      movel([0.391008, -1.437717, -2.526713, -0.747959, 1.570796, 1.961804],accel_mss,speed_ms,0,blend_radius_m)
      movel([0.391013, -1.437236, -2.527093, -0.748060, 1.570796, 1.961809],accel_mss,speed_ms,0,blend_radius_m)
      movel([0.391046, -1.436198, -2.527912, -0.748279, 1.570796, 1.961842],accel_mss,speed_ms,0,blend_radius_m)
      movel([0.391091, -1.435157, -2.528733, -0.748500, 1.570796, 1.961887],accel_mss,speed_ms,0,blend_radius_m)
      movel([0.391149, -1.434110, -2.529556, -0.748724, 1.570796, 1.961945],accel_mss,speed_ms,0,blend_radius_m)
      movel([0.391230, -1.432906, -2.530500, -0.748983, 1.570796, 1.962026],accel_mss,speed_ms,0,blend_radius_m)
      movel([0.391323, -1.431698, -2.531445, -0.749246, 1.570796, 1.962119],accel_mss,speed_ms,0,blend_radius_m)
      movel([0.391429, -1.430482, -2.532395, -0.749512, 1.570796, 1.962226],accel_mss,speed_ms,0,blend_radius_m)
      movel([0.391551, -1.429259, -2.533347, -0.749782, 1.570796, 1.962348],accel_mss,speed_ms,0,blend_radius_m)
      movel([0.391688, -1.428032, -2.534301, -0.750056, 1.570796, 1.962484],accel_mss,speed_ms,0,blend_radius_m)
      movel([0.391837, -1.426799, -2.535257, -0.750333, 1.570796, 1.962634],accel_mss,speed_ms,0,blend_radius_m)
      movel([0.392000, -1.425405, -2.536335, -0.750649, 1.570796, 1.962797],accel_mss,speed_ms,0,blend_radius_m)
      movel([0.392135, -1.424015, -2.537407, -0.750967, 1.570796, 1.962931],accel_mss,speed_ms,0,blend_radius_m)
      movel([0.392245, -1.422628, -2.538474, -0.751287, 1.570796, 1.963042],accel_mss,speed_ms,0,blend_radius_m)
      movel([0.392325, -1.421249, -2.539532, -0.751608, 1.570796, 1.963121],accel_mss,speed_ms,0,blend_radius_m)
      movel([0.392346, -1.420560, -2.540059, -0.751770, 1.570796, 1.963143],accel_mss,speed_ms,0,blend_radius_m)
      movel([0.392346, -1.419880, -2.540579, -0.751930, 1.570796, 1.963143],accel_mss,speed_ms,0,blend_radius_m)
      movel([0.392325, -1.419207, -2.541092, -0.752089, 1.570796, 1.963121],accel_mss,speed_ms,0,blend_radius_m)
      movel([0.392281, -1.418541, -2.541601, -0.752247, 1.570796, 1.963077],accel_mss,speed_ms,0,blend_radius_m)
      movel([0.392215, -1.417882, -2.542102, -0.752405, 1.570796, 1.963012],accel_mss,speed_ms,0,blend_radius_m)
      movel([0.392127, -1.417234, -2.542595, -0.752560, 1.570796, 1.962924],accel_mss,speed_ms,0,blend_radius_m)
      movel([0.392031, -1.416697, -2.543003, -0.752689, 1.570796, 1.962828],accel_mss,speed_ms,0,blend_radius_m)
      movel([0.391914, -1.416172, -2.543402, -0.752815, 1.570796, 1.962711],accel_mss,speed_ms,0,blend_radius_m)
      movel([0.391773, -1.415658, -2.543791, -0.752940, 1.570796, 1.962569],accel_mss,speed_ms,0,blend_radius_m)
      movel([0.391607, -1.415156, -2.544171, -0.753062, 1.570796, 1.962404],accel_mss,speed_ms,0,blend_radius_m)
      movel([0.391419, -1.414665, -2.544543, -0.753181, 1.570796, 1.962216],accel_mss,speed_ms,0,blend_radius_m)
      movel([0.391209, -1.414190, -2.544902, -0.753297, 1.570796, 1.962005],accel_mss,speed_ms,0,blend_radius_m)
      movel([0.390979, -1.413733, -2.545247, -0.753409, 1.570796, 1.961776],accel_mss,speed_ms,0,blend_radius_m)
      movel([0.390725, -1.413291, -2.545580, -0.753517, 1.570796, 1.961521],accel_mss,speed_ms,0,blend_radius_m)
      movel([0.390449, -1.412863, -2.545903, -0.753623, 1.570796, 1.961245],accel_mss,speed_ms,0,blend_radius_m)
      movel([0.390149, -1.412454, -2.546211, -0.753724, 1.570796, 1.960945],accel_mss,speed_ms,0,blend_radius_m)
      movel([0.389829, -1.412060, -2.546508, -0.753821, 1.570796, 1.960625],accel_mss,speed_ms,0,blend_radius_m)
      movel([0.389486, -1.411681, -2.546793, -0.753915, 1.570796, 1.960283],accel_mss,speed_ms,0,blend_radius_m)
      movel([0.389035, -1.411243, -2.547122, -0.754024, 1.570796, 1.959831],accel_mss,speed_ms,0,blend_radius_m)
      movel([0.388548, -1.410836, -2.547428, -0.754125, 1.570796, 1.959344],accel_mss,speed_ms,0,blend_radius_m)
      movel([0.388004, -1.410440, -2.547725, -0.754224, 1.570796, 1.958800],accel_mss,speed_ms,0,blend_radius_m)
      movel([0.387428, -1.410075, -2.547998, -0.754316, 1.570796, 1.958225],accel_mss,speed_ms,0,blend_radius_m)
      movel([0.386840, -1.409745, -2.548245, -0.754398, 1.570796, 1.957636],accel_mss,speed_ms,0,blend_radius_m)
      movel([0.386219, -1.409448, -2.548468, -0.754473, 1.570796, 1.957016],accel_mss,speed_ms,0,blend_radius_m)
      movel([0.385828, -1.409285, -2.548590, -0.754514, 1.570796, 1.956624],accel_mss,speed_ms,0,blend_radius_m)
      movel([0.385423, -1.409139, -2.548699, -0.754551, 1.570796, 1.956219],accel_mss,speed_ms,0,blend_radius_m)
      movel([0.385006, -1.409009, -2.548796, -0.754584, 1.570796, 1.955802],accel_mss,speed_ms,0,blend_radius_m)
      movel([0.383851, -1.408685, -2.549039, -0.754665, 1.570796, 1.954647],accel_mss,speed_ms,0,blend_radius_m)
      movel([0.383532, -1.409238, -2.548625, -0.754526, 1.570796, 1.954329],accel_mss,speed_ms,0,blend_radius_m)
      movel([0.383126, -1.409975, -2.548073, -0.754341, 1.570796, 1.953923],accel_mss,speed_ms,0,blend_radius_m)
      movel([0.381046, -1.414103, -2.544967, -0.753318, 1.570796, 1.951842],accel_mss,speed_ms,0,blend_radius_m)
      movel([0.381019, -1.414157, -2.544927, -0.753305, 1.570796, 1.951816],accel_mss,speed_ms,0,blend_radius_m)
      movel([0.380984, -1.414209, -2.544887, -0.753292, 1.570796, 1.951781],accel_mss,speed_ms,0,blend_radius_m)
      movel([0.380941, -1.414259, -2.544850, -0.753280, 1.570796, 1.951738],accel_mss,speed_ms,0,blend_radius_m)
      movel([0.380899, -1.414296, -2.544822, -0.753271, 1.570796, 1.951696],accel_mss,speed_ms,0,blend_radius_m)
      movel([0.380850, -1.414325, -2.544800, -0.753264, 1.570796, 1.951646],accel_mss,speed_ms,0,blend_radius_m)
      movel([0.380798, -1.414343, -2.544787, -0.753260, 1.570796, 1.951594],accel_mss,speed_ms,0,blend_radius_m)
      movel([0.380720, -1.414359, -2.544774, -0.753256, 1.570796, 1.951516],accel_mss,speed_ms,0,blend_radius_m)
      movel([0.380641, -1.414367, -2.544768, -0.753254, 1.570796, 1.951438],accel_mss,speed_ms,0,blend_radius_m)
      movel([0.380568, -1.414366, -2.544769, -0.753254, 1.570796, 1.951365],accel_mss,speed_ms,0,blend_radius_m)
      movel([0.380337, -1.414350, -2.544781, -0.753258, 1.570796, 1.951133],accel_mss,speed_ms,0,blend_radius_m)
      movel([0.380108, -1.414330, -2.544796, -0.753263, 1.570796, 1.950904],accel_mss,speed_ms,0,blend_radius_m)
      movel([0.377696, -1.414133, -2.544945, -0.753311, 1.570796, 1.948493],accel_mss,speed_ms,0,blend_radius_m)
      movel([0.377544, -1.414147, -2.544935, -0.753308, 1.570796, 1.948341],accel_mss,speed_ms,0,blend_radius_m)
      movel([0.377385, -1.414188, -2.544903, -0.753297, 1.570796, 1.948181],accel_mss,speed_ms,0,blend_radius_m)
      movel([0.377316, -1.414222, -2.544878, -0.753289, 1.570796, 1.948112],accel_mss,speed_ms,0,blend_radius_m)
      movel([0.377256, -1.414274, -2.544838, -0.753277, 1.570796, 1.948053],accel_mss,speed_ms,0,blend_radius_m)
      movel([0.377217, -1.414337, -2.544791, -0.753261, 1.570796, 1.948013],accel_mss,speed_ms,0,blend_radius_m)
      movel([0.377159, -1.414466, -2.544693, -0.753230, 1.570796, 1.947956],accel_mss,speed_ms,0,blend_radius_m)
      movel([0.377090, -1.414598, -2.544594, -0.753197, 1.570796, 1.947886],accel_mss,speed_ms,0,blend_radius_m)
      movel([0.377010, -1.414725, -2.544497, -0.753166, 1.570796, 1.947807],accel_mss,speed_ms,0,blend_radius_m)
      movel([0.376921, -1.414851, -2.544402, -0.753136, 1.570796, 1.947717],accel_mss,speed_ms,0,blend_radius_m)
      movel([0.376332, -1.415635, -2.543809, -0.752945, 1.570796, 1.947129],accel_mss,speed_ms,0,blend_radius_m)
      movel([0.375736, -1.416416, -2.543217, -0.752757, 1.570796, 1.946533],accel_mss,speed_ms,0,blend_radius_m)
      movel([0.375083, -1.417257, -2.542578, -0.752554, 1.570796, 1.945880],accel_mss,speed_ms,0,blend_radius_m)
      movel([0.374421, -1.418095, -2.541941, -0.752354, 1.570796, 1.945218],accel_mss,speed_ms,0,blend_radius_m)
      movel([0.373801, -1.418859, -2.541359, -0.752172, 1.570796, 1.944597],accel_mss,speed_ms,0,blend_radius_m)
      movel([0.373169, -1.419616, -2.540781, -0.751993, 1.570796, 1.943965],accel_mss,speed_ms,0,blend_radius_m)
      movel([0.372591, -1.420290, -2.540265, -0.751833, 1.570796, 1.943387],accel_mss,speed_ms,0,blend_radius_m)
      movel([0.372002, -1.420960, -2.539753, -0.751676, 1.570796, 1.942799],accel_mss,speed_ms,0,blend_radius_m)
      movel([0.371402, -1.421622, -2.539246, -0.751521, 1.570796, 1.942199],accel_mss,speed_ms,0,blend_radius_m)
      movel([0.370791, -1.422279, -2.538742, -0.751368, 1.570796, 1.941588],accel_mss,speed_ms,0,blend_radius_m)
      movel([0.370171, -1.422927, -2.538244, -0.751218, 1.570796, 1.940968],accel_mss,speed_ms,0,blend_radius_m)
      movel([0.369539, -1.423568, -2.537751, -0.751070, 1.570796, 1.940336],accel_mss,speed_ms,0,blend_radius_m)
      movel([0.368900, -1.424201, -2.537264, -0.750924, 1.570796, 1.939697],accel_mss,speed_ms,0,blend_radius_m)
      movel([0.368252, -1.424827, -2.536781, -0.750781, 1.570796, 1.939048],accel_mss,speed_ms,0,blend_radius_m)
      movel([0.367591, -1.425445, -2.536304, -0.750640, 1.570796, 1.938388],accel_mss,speed_ms,0,blend_radius_m)
      movel([0.366924, -1.426056, -2.535832, -0.750501, 1.570796, 1.937720],accel_mss,speed_ms,0,blend_radius_m)
      movel([0.366244, -1.426659, -2.535366, -0.750365, 1.570796, 1.937041],accel_mss,speed_ms,0,blend_radius_m)
      movel([0.365557, -1.427255, -2.534904, -0.750230, 1.570796, 1.936354],accel_mss,speed_ms,0,blend_radius_m)
      movel([0.364862, -1.427840, -2.534450, -0.750099, 1.570796, 1.935659],accel_mss,speed_ms,0,blend_radius_m)
      movel([0.364160, -1.428418, -2.534002, -0.749970, 1.570796, 1.934957],accel_mss,speed_ms,0,blend_radius_m)
      movel([0.363449, -1.428986, -2.533560, -0.749843, 1.570796, 1.934245],accel_mss,speed_ms,0,blend_radius_m)
      movel([0.362732, -1.429545, -2.533125, -0.749719, 1.570796, 1.933528],accel_mss,speed_ms,0,blend_radius_m)
      movel([0.362008, -1.430092, -2.532699, -0.749598, 1.570796, 1.932805],accel_mss,speed_ms,0,blend_radius_m)
      movel([0.361278, -1.430632, -2.532278, -0.749479, 1.570796, 1.932074],accel_mss,speed_ms,0,blend_radius_m)
      movel([0.360551, -1.431154, -2.531870, -0.749364, 1.570796, 1.931347],accel_mss,speed_ms,0,blend_radius_m)
      movel([0.359817, -1.431667, -2.531470, -0.749252, 1.570796, 1.930614],accel_mss,speed_ms,0,blend_radius_m)
      movel([0.359077, -1.432169, -2.531077, -0.749143, 1.570796, 1.929874],accel_mss,speed_ms,0,blend_radius_m)
      movel([0.358332, -1.432660, -2.530693, -0.749036, 1.570796, 1.929128],accel_mss,speed_ms,0,blend_radius_m)
      movel([0.357582, -1.433140, -2.530317, -0.748932, 1.570796, 1.928379],accel_mss,speed_ms,0,blend_radius_m)
      movel([0.356828, -1.433611, -2.529947, -0.748831, 1.570796, 1.927625],accel_mss,speed_ms,0,blend_radius_m)
      movel([0.356069, -1.434070, -2.529587, -0.748732, 1.570796, 1.926865],accel_mss,speed_ms,0,blend_radius_m)
      movel([0.355306, -1.434516, -2.529236, -0.748636, 1.570796, 1.926102],accel_mss,speed_ms,0,blend_radius_m)
      movel([0.354537, -1.434953, -2.528893, -0.748543, 1.570796, 1.925333],accel_mss,speed_ms,0,blend_radius_m)
      movel([0.353788, -1.435366, -2.528568, -0.748455, 1.570796, 1.924585],accel_mss,speed_ms,0,blend_radius_m)
      movel([0.353034, -1.435767, -2.528252, -0.748370, 1.570796, 1.923830],accel_mss,speed_ms,0,blend_radius_m)
      movel([0.352277, -1.436154, -2.527947, -0.748288, 1.570796, 1.923073],accel_mss,speed_ms,0,blend_radius_m)
      movel([0.351516, -1.436531, -2.527649, -0.748208, 1.570796, 1.922312],accel_mss,speed_ms,0,blend_radius_m)
      movel([0.350754, -1.436894, -2.527363, -0.748132, 1.570796, 1.921551],accel_mss,speed_ms,0,blend_radius_m)
      movel([0.349988, -1.437243, -2.527088, -0.748058, 1.570796, 1.920784],accel_mss,speed_ms,0,blend_radius_m)
      movel([0.349222, -1.437580, -2.526821, -0.747988, 1.570796, 1.920018],accel_mss,speed_ms,0,blend_radius_m)
      movel([0.348452, -1.437905, -2.526565, -0.747920, 1.570796, 1.919249],accel_mss,speed_ms,0,blend_radius_m)
      movel([0.347682, -1.438215, -2.526319, -0.747855, 1.570796, 1.918479],accel_mss,speed_ms,0,blend_radius_m)
      movel([0.346942, -1.438501, -2.526093, -0.747796, 1.570796, 1.917738],accel_mss,speed_ms,0,blend_radius_m)
      movel([0.346197, -1.438776, -2.525874, -0.747738, 1.570796, 1.916993],accel_mss,speed_ms,0,blend_radius_m)
      movel([0.345456, -1.439037, -2.525667, -0.747684, 1.570796, 1.916252],accel_mss,speed_ms,0,blend_radius_m)
      movel([0.344712, -1.439289, -2.525468, -0.747632, 1.570796, 1.915508],accel_mss,speed_ms,0,blend_radius_m)
      movel([0.343967, -1.439527, -2.525279, -0.747583, 1.570796, 1.914764],accel_mss,speed_ms,0,blend_radius_m)
      movel([0.343243, -1.439745, -2.525106, -0.747538, 1.570796, 1.914040],accel_mss,speed_ms,0,blend_radius_m)
      movel([0.342517, -1.439952, -2.524941, -0.747495, 1.570796, 1.913314],accel_mss,speed_ms,0,blend_radius_m)
      movel([0.341795, -1.440145, -2.524788, -0.747456, 1.570796, 1.912591],accel_mss,speed_ms,0,blend_radius_m)
      movel([0.341071, -1.440326, -2.524644, -0.747419, 1.570796, 1.911867],accel_mss,speed_ms,0,blend_radius_m)
      movel([0.340352, -1.440493, -2.524512, -0.747384, 1.570796, 1.911149],accel_mss,speed_ms,0,blend_radius_m)
      movel([0.339621, -1.440649, -2.524388, -0.747352, 1.570796, 1.910417],accel_mss,speed_ms,0,blend_radius_m)
      movel([0.338890, -1.440790, -2.524275, -0.747323, 1.570796, 1.909687],accel_mss,speed_ms,0,blend_radius_m)
      movel([0.338165, -1.440920, -2.524172, -0.747297, 1.570796, 1.908961],accel_mss,speed_ms,0,blend_radius_m)
      movel([0.337442, -1.441036, -2.524080, -0.747273, 1.570796, 1.908238],accel_mss,speed_ms,0,blend_radius_m)
      movel([0.336723, -1.441138, -2.523999, -0.747252, 1.570796, 1.907519],accel_mss,speed_ms,0,blend_radius_m)
      movel([0.335963, -1.441234, -2.523922, -0.747233, 1.570796, 1.906759],accel_mss,speed_ms,0,blend_radius_m)
      movel([0.335208, -1.441316, -2.523857, -0.747216, 1.570796, 1.906004],accel_mss,speed_ms,0,blend_radius_m)
      movel([0.334457, -1.441386, -2.523801, -0.747202, 1.570796, 1.905253],accel_mss,speed_ms,0,blend_radius_m)
      movel([0.333710, -1.441447, -2.523753, -0.747189, 1.570796, 1.904507],accel_mss,speed_ms,0,blend_radius_m)
      movel([0.332967, -1.441493, -2.523716, -0.747180, 1.570796, 1.903763],accel_mss,speed_ms,0,blend_radius_m)
      movel([0.329715, -1.441675, -2.523571, -0.747143, 1.570796, 1.900511],accel_mss,speed_ms,0,blend_radius_m)
      movel([0.329386, -1.442137, -2.523203, -0.747049, 1.570796, 1.900182],accel_mss,speed_ms,0,blend_radius_m)
      movel([0.329307, -1.442240, -2.523121, -0.747029, 1.570796, 1.900104],accel_mss,speed_ms,0,blend_radius_m)
      movel([0.329218, -1.442336, -2.523044, -0.747009, 1.570796, 1.900015],accel_mss,speed_ms,0,blend_radius_m)
      movel([0.329123, -1.442425, -2.522973, -0.746991, 1.570796, 1.899919],accel_mss,speed_ms,0,blend_radius_m)
      movel([0.329019, -1.442510, -2.522905, -0.746974, 1.570796, 1.899815],accel_mss,speed_ms,0,blend_radius_m)
      movel([0.328913, -1.442580, -2.522849, -0.746960, 1.570796, 1.899710],accel_mss,speed_ms,0,blend_radius_m)
      movel([0.328802, -1.442642, -2.522799, -0.746947, 1.570796, 1.899598],accel_mss,speed_ms,0,blend_radius_m)
      movel([0.328694, -1.442690, -2.522761, -0.746938, 1.570796, 1.899490],accel_mss,speed_ms,0,blend_radius_m)
      movel([0.328584, -1.442725, -2.522734, -0.746931, 1.570796, 1.899380],accel_mss,speed_ms,0,blend_radius_m)
      movel([0.328442, -1.442758, -2.522707, -0.746924, 1.570796, 1.899238],accel_mss,speed_ms,0,blend_radius_m)
      movel([0.328305, -1.442780, -2.522690, -0.746920, 1.570796, 1.899101],accel_mss,speed_ms,0,blend_radius_m)
      movel([0.328168, -1.442793, -2.522679, -0.746917, 1.570796, 1.898964],accel_mss,speed_ms,0,blend_radius_m)
      movel([0.328036, -1.442794, -2.522678, -0.746917, 1.570796, 1.898832],accel_mss,speed_ms,0,blend_radius_m)
      movel([0.323844, -1.442695, -2.522758, -0.746937, 1.570796, 1.894641],accel_mss,speed_ms,0,blend_radius_m)
      movel([0.321918, -1.442649, -2.522794, -0.746946, 1.570796, 1.892714],accel_mss,speed_ms,0,blend_radius_m)
      movel([0.319994, -1.442597, -2.522836, -0.746956, 1.570796, 1.890790],accel_mss,speed_ms,0,blend_radius_m)
      movel([0.319329, -1.442571, -2.522856, -0.746962, 1.570796, 1.890125],accel_mss,speed_ms,0,blend_radius_m)
      movel([0.318669, -1.442535, -2.522885, -0.746969, 1.570796, 1.889465],accel_mss,speed_ms,0,blend_radius_m)
      movel([0.318013, -1.442490, -2.522921, -0.746978, 1.570796, 1.888809],accel_mss,speed_ms,0,blend_radius_m)
      movel([0.317850, -1.442468, -2.522939, -0.746983, 1.570796, 1.888646],accel_mss,speed_ms,0,blend_radius_m)
      movel([0.317697, -1.442429, -2.522970, -0.746990, 1.570796, 1.888493],accel_mss,speed_ms,0,blend_radius_m)
      movel([0.317553, -1.442377, -2.523011, -0.747001, 1.570796, 1.888349],accel_mss,speed_ms,0,blend_radius_m)
      movel([0.317424, -1.442309, -2.523065, -0.747015, 1.570796, 1.888220],accel_mss,speed_ms,0,blend_radius_m)
      movel([0.317355, -1.442253, -2.523110, -0.747026, 1.570796, 1.888151],accel_mss,speed_ms,0,blend_radius_m)
      movel([0.317298, -1.442186, -2.523163, -0.747039, 1.570796, 1.888095],accel_mss,speed_ms,0,blend_radius_m)
      movel([0.317262, -1.442106, -2.523227, -0.747056, 1.570796, 1.888058],accel_mss,speed_ms,0,blend_radius_m)
      movel([0.317241, -1.442017, -2.523299, -0.747074, 1.570796, 1.888038],accel_mss,speed_ms,0,blend_radius_m)
      movel([0.317241, -1.441920, -2.523376, -0.747093, 1.570796, 1.888037],accel_mss,speed_ms,0,blend_radius_m)
      movel([0.317266, -1.441727, -2.523529, -0.747133, 1.570796, 1.888062],accel_mss,speed_ms,0,blend_radius_m)
      movel([0.317307, -1.441531, -2.523686, -0.747172, 1.570796, 1.888103],accel_mss,speed_ms,0,blend_radius_m)
      movel([0.317366, -1.441332, -2.523844, -0.747213, 1.570796, 1.888162],accel_mss,speed_ms,0,blend_radius_m)
      movel([0.317441, -1.441131, -2.524004, -0.747254, 1.570796, 1.888237],accel_mss,speed_ms,0,blend_radius_m)
      movel([0.317857, -1.440156, -2.524779, -0.747453, 1.570796, 1.888653],accel_mss,speed_ms,0,blend_radius_m)
      movel([0.318288, -1.439181, -2.525553, -0.747655, 1.570796, 1.889084],accel_mss,speed_ms,0,blend_radius_m)
      movel([0.319674, -1.435971, -2.528092, -0.748327, 1.570796, 1.890471],accel_mss,speed_ms,0,blend_radius_m)
      movel([0.319898, -1.435346, -2.528583, -0.748459, 1.570796, 1.890694],accel_mss,speed_ms,0,blend_radius_m)
      movel([0.318917, -1.435409, -2.528534, -0.748446, 1.570796, 1.889714],accel_mss,speed_ms,0,blend_radius_m)
      movel([0.317936, -1.435473, -2.528483, -0.748432, 1.570796, 1.888733],accel_mss,speed_ms,0,blend_radius_m)
      movel([0.315692, -1.441850, -2.523431, -0.747108, 1.570796, 1.886489],accel_mss,speed_ms,0,blend_radius_m)
      movel([0.314773, -1.444460, -2.521346, -0.746583, 1.570796, 1.885569],accel_mss,speed_ms,0,blend_radius_m)
      movel([0.313846, -1.447061, -2.519257, -0.746071, 1.570796, 1.884642],accel_mss,speed_ms,0,blend_radius_m)
      movel([0.313754, -1.447292, -2.519071, -0.746026, 1.570796, 1.884550],accel_mss,speed_ms,0,blend_radius_m)
      movel([0.313650, -1.447523, -2.518885, -0.745981, 1.570796, 1.884446],accel_mss,speed_ms,0,blend_radius_m)
      movel([0.313528, -1.447754, -2.518699, -0.745936, 1.570796, 1.884325],accel_mss,speed_ms,0,blend_radius_m)
      movel([0.313393, -1.447983, -2.518515, -0.745892, 1.570796, 1.884189],accel_mss,speed_ms,0,blend_radius_m)
      movel([0.313241, -1.448208, -2.518333, -0.745848, 1.570796, 1.884037],accel_mss,speed_ms,0,blend_radius_m)
      movel([0.313169, -1.448302, -2.518257, -0.745830, 1.570796, 1.883966],accel_mss,speed_ms,0,blend_radius_m)
      movel([0.313084, -1.448391, -2.518185, -0.745813, 1.570796, 1.883881],accel_mss,speed_ms,0,blend_radius_m)
      movel([0.312991, -1.448475, -2.518117, -0.745797, 1.570796, 1.883787],accel_mss,speed_ms,0,blend_radius_m)
      movel([0.312890, -1.448550, -2.518057, -0.745782, 1.570796, 1.883686],accel_mss,speed_ms,0,blend_radius_m)
      movel([0.312781, -1.448614, -2.518005, -0.745770, 1.570796, 1.883577],accel_mss,speed_ms,0,blend_radius_m)
      movel([0.312669, -1.448670, -2.517960, -0.745759, 1.570796, 1.883466],accel_mss,speed_ms,0,blend_radius_m)
      movel([0.312558, -1.448711, -2.517927, -0.745751, 1.570796, 1.883355],accel_mss,speed_ms,0,blend_radius_m)
      movel([0.312444, -1.448742, -2.517902, -0.745745, 1.570796, 1.883241],accel_mss,speed_ms,0,blend_radius_m)
      movel([0.312092, -1.448811, -2.517846, -0.745732, 1.570796, 1.882888],accel_mss,speed_ms,0,blend_radius_m)
      movel([0.311740, -1.448872, -2.517797, -0.745720, 1.570796, 1.882536],accel_mss,speed_ms,0,blend_radius_m)
      movel([0.311392, -1.448920, -2.517758, -0.745711, 1.570796, 1.882188],accel_mss,speed_ms,0,blend_radius_m)
      movel([0.311046, -1.448959, -2.517726, -0.745704, 1.570796, 1.881842],accel_mss,speed_ms,0,blend_radius_m)
      movel([0.310704, -1.448986, -2.517705, -0.745698, 1.570796, 1.881500],accel_mss,speed_ms,0,blend_radius_m)
      movel([0.308856, -1.449110, -2.517604, -0.745675, 1.570796, 1.879653],accel_mss,speed_ms,0,blend_radius_m)
      movel([0.307890, -1.451920, -2.515327, -0.745142, 1.570796, 1.878686],accel_mss,speed_ms,0,blend_radius_m)
      movel([0.306930, -1.454717, -2.513049, -0.744623, 1.570796, 1.877726],accel_mss,speed_ms,0,blend_radius_m)
      movel([0.321643, -1.458076, -2.510297, -0.744016, 1.570796, 1.892440],accel_mss,speed_ms,0,blend_radius_m)
      movel([0.327249, -1.459428, -2.509184, -0.743777, 1.570796, 1.898045],accel_mss,speed_ms,0,blend_radius_m)
      movel([0.331985, -1.460602, -2.508216, -0.743571, 1.570796, 1.902781],accel_mss,speed_ms,0,blend_radius_m)
      movel([0.336201, -1.461671, -2.507332, -0.743386, 1.570796, 1.906997],accel_mss,speed_ms,0,blend_radius_m)
      movel([0.336481, -1.461719, -2.507292, -0.743378, 1.570796, 1.907277],accel_mss,speed_ms,0,blend_radius_m)
      movel([0.336565, -1.461686, -2.507319, -0.743383, 1.570796, 1.907361],accel_mss,speed_ms,0,blend_radius_m)
      movel([0.336663, -1.461615, -2.507378, -0.743396, 1.570796, 1.907460],accel_mss,speed_ms,0,blend_radius_m)
      movel([0.336752, -1.461531, -2.507448, -0.743410, 1.570796, 1.907549],accel_mss,speed_ms,0,blend_radius_m)
      movel([0.336997, -1.461218, -2.507707, -0.743464, 1.570796, 1.907793],accel_mss,speed_ms,0,blend_radius_m)
      movel([0.337381, -1.460630, -2.508193, -0.743566, 1.570796, 1.908177],accel_mss,speed_ms,0,blend_radius_m)
      movel([0.337671, -1.460183, -2.508561, -0.743644, 1.570796, 1.908467],accel_mss,speed_ms,0,blend_radius_m)
      movel([0.337804, -1.459986, -2.508724, -0.743679, 1.570796, 1.908601],accel_mss,speed_ms,0,blend_radius_m)
      movel([0.337943, -1.459793, -2.508883, -0.743713, 1.570796, 1.908739],accel_mss,speed_ms,0,blend_radius_m)
      movel([0.338182, -1.459473, -2.509147, -0.743769, 1.570796, 1.908978],accel_mss,speed_ms,0,blend_radius_m)
      movel([0.338208, -1.459442, -2.509172, -0.743774, 1.570796, 1.909005],accel_mss,speed_ms,0,blend_radius_m)
      movel([0.338242, -1.459415, -2.509195, -0.743779, 1.570796, 1.909038],accel_mss,speed_ms,0,blend_radius_m)
      movel([0.338277, -1.459394, -2.509212, -0.743783, 1.570796, 1.909074],accel_mss,speed_ms,0,blend_radius_m)
      movel([0.338400, -1.459338, -2.509258, -0.743793, 1.570796, 1.909197],accel_mss,speed_ms,0,blend_radius_m)
      movel([0.338523, -1.459294, -2.509295, -0.743800, 1.570796, 1.909319],accel_mss,speed_ms,0,blend_radius_m)
      movel([0.338648, -1.459260, -2.509323, -0.743807, 1.570796, 1.909445],accel_mss,speed_ms,0,blend_radius_m)
      movel([0.343772, -1.458166, -2.510223, -0.744000, 1.570796, 1.914568],accel_mss,speed_ms,0,blend_radius_m)
      movel([0.348794, -1.457117, -2.511085, -0.744188, 1.570796, 1.919590],accel_mss,speed_ms,0,blend_radius_m)
      movel([0.348995, -1.457081, -2.511114, -0.744194, 1.570796, 1.919791],accel_mss,speed_ms,0,blend_radius_m)
      movel([0.349193, -1.457058, -2.511133, -0.744198, 1.570796, 1.919989],accel_mss,speed_ms,0,blend_radius_m)
      movel([0.349389, -1.457046, -2.511142, -0.744200, 1.570796, 1.920185],accel_mss,speed_ms,0,blend_radius_m)
      movel([0.349479, -1.457050, -2.511140, -0.744200, 1.570796, 1.920275],accel_mss,speed_ms,0,blend_radius_m)
      movel([0.349560, -1.457063, -2.511128, -0.744197, 1.570796, 1.920357],accel_mss,speed_ms,0,blend_radius_m)
      movel([0.349638, -1.457089, -2.511107, -0.744193, 1.570796, 1.920434],accel_mss,speed_ms,0,blend_radius_m)
      movel([0.351833, -1.458041, -2.510325, -0.744022, 1.570796, 1.922629],accel_mss,speed_ms,0,blend_radius_m)
      movel([0.353078, -1.458589, -2.509875, -0.743925, 1.570796, 1.923875],accel_mss,speed_ms,0,blend_radius_m)
      movel([0.354315, -1.459145, -2.509417, -0.743827, 1.570796, 1.925111],accel_mss,speed_ms,0,blend_radius_m)
      movel([0.355751, -1.459804, -2.508874, -0.743711, 1.570796, 1.926547],accel_mss,speed_ms,0,blend_radius_m)
      movel([0.357181, -1.460468, -2.508327, -0.743595, 1.570796, 1.927977],accel_mss,speed_ms,0,blend_radius_m)
      movel([0.364532, -1.463955, -2.505438, -0.742996, 1.570796, 1.935329],accel_mss,speed_ms,0,blend_radius_m)
      movel([0.364147, -1.464542, -2.504950, -0.742897, 1.570796, 1.934944],accel_mss,speed_ms,0,blend_radius_m)
      movel([0.360132, -1.470721, -2.499780, -0.741888, 1.570796, 1.930928],accel_mss,speed_ms,0,blend_radius_m)
      movel([0.359272, -1.472034, -2.498674, -0.741681, 1.570796, 1.930068],accel_mss,speed_ms,0,blend_radius_m)
      movel([0.358506, -1.473198, -2.497691, -0.741500, 1.570796, 1.929302],accel_mss,speed_ms,0,blend_radius_m)
      movel([0.358478, -1.473230, -2.497664, -0.741495, 1.570796, 1.929275],accel_mss,speed_ms,0,blend_radius_m)
      movel([0.358446, -1.473258, -2.497641, -0.741491, 1.570796, 1.929243],accel_mss,speed_ms,0,blend_radius_m)
      movel([0.358424, -1.473268, -2.497632, -0.741489, 1.570796, 1.929220],accel_mss,speed_ms,0,blend_radius_m)
      movel([0.358402, -1.473270, -2.497630, -0.741489, 1.570796, 1.929198],accel_mss,speed_ms,0,blend_radius_m)
      movel([0.358383, -1.473264, -2.497635, -0.741490, 1.570796, 1.929179],accel_mss,speed_ms,0,blend_radius_m)
      movel([0.357147, -1.472418, -2.498350, -0.741621, 1.570796, 1.927943],accel_mss,speed_ms,0,blend_radius_m)
      movel([0.356454, -1.471942, -2.498752, -0.741695, 1.570796, 1.927250],accel_mss,speed_ms,0,blend_radius_m)
      movel([0.355765, -1.471462, -2.499156, -0.741771, 1.570796, 1.926561],accel_mss,speed_ms,0,blend_radius_m)
      movel([0.354136, -1.470317, -2.500120, -0.741952, 1.570796, 1.924932],accel_mss,speed_ms,0,blend_radius_m)
      movel([0.352498, -1.469178, -2.501076, -0.742134, 1.570796, 1.923294],accel_mss,speed_ms,0,blend_radius_m)
      movel([0.351087, -1.468242, -2.501862, -0.742286, 1.570796, 1.921883],accel_mss,speed_ms,0,blend_radius_m)
      movel([0.349797, -1.467428, -2.502543, -0.742418, 1.570796, 1.920593],accel_mss,speed_ms,0,blend_radius_m)
      movel([0.349754, -1.467437, -2.502535, -0.742417, 1.570796, 1.920550],accel_mss,speed_ms,0,blend_radius_m)
      movel([0.349713, -1.467460, -2.502516, -0.742413, 1.570796, 1.920510],accel_mss,speed_ms,0,blend_radius_m)
      movel([0.349617, -1.467544, -2.502445, -0.742399, 1.570796, 1.920413],accel_mss,speed_ms,0,blend_radius_m)
      movel([0.349532, -1.467639, -2.502366, -0.742384, 1.570796, 1.920328],accel_mss,speed_ms,0,blend_radius_m)
      movel([0.349462, -1.467739, -2.502282, -0.742367, 1.570796, 1.920258],accel_mss,speed_ms,0,blend_radius_m)
      movel([0.344256, -1.476421, -2.494959, -0.741009, 1.570796, 1.915053],accel_mss,speed_ms,0,blend_radius_m)
      movel([0.344252, -1.476475, -2.494912, -0.741001, 1.570796, 1.915048],accel_mss,speed_ms,0,blend_radius_m)
      movel([0.344270, -1.476520, -2.494875, -0.740995, 1.570796, 1.915067],accel_mss,speed_ms,0,blend_radius_m)
      movel([0.344294, -1.476539, -2.494859, -0.740992, 1.570796, 1.915091],accel_mss,speed_ms,0,blend_radius_m)
      movel([0.344333, -1.476539, -2.494858, -0.740992, 1.570796, 1.915130],accel_mss,speed_ms,0,blend_radius_m)
      movel([0.348677, -1.475673, -2.495594, -0.741122, 1.570796, 1.919474],accel_mss,speed_ms,0,blend_radius_m)
      movel([0.353320, -1.474728, -2.496396, -0.741265, 1.570796, 1.924117],accel_mss,speed_ms,0,blend_radius_m)
      movel([0.355242, -1.474345, -2.496720, -0.741323, 1.570796, 1.926039],accel_mss,speed_ms,0,blend_radius_m)
      movel([0.356189, -1.474167, -2.496872, -0.741351, 1.570796, 1.926986],accel_mss,speed_ms,0,blend_radius_m)
      movel([0.357134, -1.474000, -2.497012, -0.741376, 1.570796, 1.927930],accel_mss,speed_ms,0,blend_radius_m)
      movel([0.357714, -1.473906, -2.497092, -0.741391, 1.570796, 1.928510],accel_mss,speed_ms,0,blend_radius_m)
      movel([0.358290, -1.473822, -2.497163, -0.741404, 1.570796, 1.929086],accel_mss,speed_ms,0,blend_radius_m)
      movel([0.358331, -1.473824, -2.497162, -0.741403, 1.570796, 1.929128],accel_mss,speed_ms,0,blend_radius_m)
      movel([0.358364, -1.473837, -2.497151, -0.741401, 1.570796, 1.929160],accel_mss,speed_ms,0,blend_radius_m)
      movel([0.358385, -1.473862, -2.497129, -0.741397, 1.570796, 1.929181],accel_mss,speed_ms,0,blend_radius_m)
      movel([0.358392, -1.473897, -2.497100, -0.741392, 1.570796, 1.929188],accel_mss,speed_ms,0,blend_radius_m)
      movel([0.358383, -1.473935, -2.497068, -0.741386, 1.570796, 1.929179],accel_mss,speed_ms,0,blend_radius_m)
      movel([0.358320, -1.474083, -2.496943, -0.741364, 1.570796, 1.929116],accel_mss,speed_ms,0,blend_radius_m)
      movel([0.358247, -1.474228, -2.496819, -0.741341, 1.570796, 1.929043],accel_mss,speed_ms,0,blend_radius_m)
      movel([0.358166, -1.474374, -2.496696, -0.741319, 1.570796, 1.928962],accel_mss,speed_ms,0,blend_radius_m)
      movel([0.358075, -1.474518, -2.496574, -0.741297, 1.570796, 1.928871],accel_mss,speed_ms,0,blend_radius_m)
      movel([0.355483, -1.478437, -2.493242, -0.740711, 1.570796, 1.926279],accel_mss,speed_ms,0,blend_radius_m)
      movel([0.352786, -1.482515, -2.489748, -0.740126, 1.570796, 1.923582],accel_mss,speed_ms,0,blend_radius_m)
      movel([0.352759, -1.482546, -2.489721, -0.740122, 1.570796, 1.923555],accel_mss,speed_ms,0,blend_radius_m)
      movel([0.352726, -1.482572, -2.489699, -0.740118, 1.570796, 1.923523],accel_mss,speed_ms,0,blend_radius_m)
      movel([0.352688, -1.482590, -2.489683, -0.740116, 1.570796, 1.923484],accel_mss,speed_ms,0,blend_radius_m)
      movel([0.352650, -1.482596, -2.489678, -0.740115, 1.570796, 1.923447],accel_mss,speed_ms,0,blend_radius_m)
      movel([0.349127, -1.483333, -2.489044, -0.740012, 1.570796, 1.919923],accel_mss,speed_ms,0,blend_radius_m)
      speed_ms = 0.003
      movel([0.349127, -1.486320, -2.490369, -0.735700, 1.570796, 1.919923],accel_mss,speed_ms,0,blend_radius_m)
      speed_ms = 0.007
      movel([0.329121, -1.490727, -2.486541, -0.735122, 1.570796, 1.899918],accel_mss,speed_ms,0,blend_radius_m)
      movel([0.326624, -1.487389, -2.489443, -0.735557, 1.570796, 1.897421],accel_mss,speed_ms,0,blend_radius_m)
      movel([0.324102, -1.484049, -2.492329, -0.736010, 1.570796, 1.894899],accel_mss,speed_ms,0,blend_radius_m)
      movel([0.325153, -1.482426, -2.493726, -0.736237, 1.570796, 1.895949],accel_mss,speed_ms,0,blend_radius_m)
      movel([0.326209, -1.480800, -2.495121, -0.736468, 1.570796, 1.897005],accel_mss,speed_ms,0,blend_radius_m)
      movel([0.325032, -1.480531, -2.495351, -0.736507, 1.570796, 1.895828],accel_mss,speed_ms,0,blend_radius_m)
      movel([0.324303, -1.480374, -2.495485, -0.736530, 1.570796, 1.895099],accel_mss,speed_ms,0,blend_radius_m)
      movel([0.315110, -1.478630, -2.496976, -0.736783, 1.570796, 1.885906],accel_mss,speed_ms,0,blend_radius_m)
      movel([0.311619, -1.477981, -2.497529, -0.736879, 1.570796, 1.882415],accel_mss,speed_ms,0,blend_radius_m)
      movel([0.310032, -1.477680, -2.497785, -0.736924, 1.570796, 1.880828],accel_mss,speed_ms,0,blend_radius_m)
      movel([0.308452, -1.477368, -2.498051, -0.736970, 1.570796, 1.879249],accel_mss,speed_ms,0,blend_radius_m)
      movel([0.306876, -1.477047, -2.498324, -0.737018, 1.570796, 1.877673],accel_mss,speed_ms,0,blend_radius_m)
      movel([0.305660, -1.476784, -2.498548, -0.737057, 1.570796, 1.876456],accel_mss,speed_ms,0,blend_radius_m)
      movel([0.304453, -1.476509, -2.498781, -0.737098, 1.570796, 1.875249],accel_mss,speed_ms,0,blend_radius_m)
      movel([0.303253, -1.476222, -2.499025, -0.737142, 1.570796, 1.874050],accel_mss,speed_ms,0,blend_radius_m)
      movel([0.302430, -1.476016, -2.499201, -0.737173, 1.570796, 1.873226],accel_mss,speed_ms,0,blend_radius_m)
      movel([0.301614, -1.475798, -2.499386, -0.737206, 1.570796, 1.872410],accel_mss,speed_ms,0,blend_radius_m)
      movel([0.300804, -1.475572, -2.499577, -0.737240, 1.570796, 1.871600],accel_mss,speed_ms,0,blend_radius_m)
      movel([0.299999, -1.475338, -2.499776, -0.737275, 1.570796, 1.870795],accel_mss,speed_ms,0,blend_radius_m)
      movel([0.299265, -1.475111, -2.499968, -0.737310, 1.570796, 1.870061],accel_mss,speed_ms,0,blend_radius_m)
      movel([0.298537, -1.474874, -2.500169, -0.737346, 1.570796, 1.869333],accel_mss,speed_ms,0,blend_radius_m)
      movel([0.297819, -1.474626, -2.500379, -0.737384, 1.570796, 1.868615],accel_mss,speed_ms,0,blend_radius_m)
      movel([0.297109, -1.474366, -2.500599, -0.737424, 1.570796, 1.867905],accel_mss,speed_ms,0,blend_radius_m)
      movel([0.296406, -1.474094, -2.500829, -0.737466, 1.570796, 1.867203],accel_mss,speed_ms,0,blend_radius_m)
      movel([0.295713, -1.473813, -2.501067, -0.737509, 1.570796, 1.866509],accel_mss,speed_ms,0,blend_radius_m)
      movel([0.295027, -1.473520, -2.501314, -0.737554, 1.570796, 1.865823],accel_mss,speed_ms,0,blend_radius_m)
      movel([0.294528, -1.473293, -2.501506, -0.737589, 1.570796, 1.865325],accel_mss,speed_ms,0,blend_radius_m)
      movel([0.294040, -1.473054, -2.501709, -0.737627, 1.570796, 1.864837],accel_mss,speed_ms,0,blend_radius_m)
      movel([0.293562, -1.472804, -2.501919, -0.737666, 1.570796, 1.864358],accel_mss,speed_ms,0,blend_radius_m)
      movel([0.293093, -1.472543, -2.502140, -0.737706, 1.570796, 1.863889],accel_mss,speed_ms,0,blend_radius_m)
      movel([0.292636, -1.472269, -2.502370, -0.737749, 1.570796, 1.863432],accel_mss,speed_ms,0,blend_radius_m)
      movel([0.292189, -1.471984, -2.502611, -0.737794, 1.570796, 1.862986],accel_mss,speed_ms,0,blend_radius_m)
      movel([0.291754, -1.471687, -2.502861, -0.737841, 1.570796, 1.862551],accel_mss,speed_ms,0,blend_radius_m)
      movel([0.291328, -1.471381, -2.503119, -0.737889, 1.570796, 1.862125],accel_mss,speed_ms,0,blend_radius_m)
      movel([0.290973, -1.471104, -2.503352, -0.737933, 1.570796, 1.861769],accel_mss,speed_ms,0,blend_radius_m)
      movel([0.290628, -1.470817, -2.503594, -0.737979, 1.570796, 1.861425],accel_mss,speed_ms,0,blend_radius_m)
      movel([0.290296, -1.470519, -2.503844, -0.738026, 1.570796, 1.861092],accel_mss,speed_ms,0,blend_radius_m)
      movel([0.289978, -1.470209, -2.504105, -0.738076, 1.570796, 1.860774],accel_mss,speed_ms,0,blend_radius_m)
      movel([0.289671, -1.469888, -2.504374, -0.738127, 1.570796, 1.860467],accel_mss,speed_ms,0,blend_radius_m)
      movel([0.289378, -1.469558, -2.504651, -0.738180, 1.570796, 1.860174],accel_mss,speed_ms,0,blend_radius_m)
      movel([0.289096, -1.469216, -2.504938, -0.738235, 1.570796, 1.859893],accel_mss,speed_ms,0,blend_radius_m)
      movel([0.288831, -1.468865, -2.505232, -0.738292, 1.570796, 1.859627],accel_mss,speed_ms,0,blend_radius_m)
      movel([0.288626, -1.468570, -2.505479, -0.738340, 1.570796, 1.859423],accel_mss,speed_ms,0,blend_radius_m)
      movel([0.288435, -1.468269, -2.505731, -0.738389, 1.570796, 1.859231],accel_mss,speed_ms,0,blend_radius_m)
      movel([0.288257, -1.467957, -2.505992, -0.738440, 1.570796, 1.859053],accel_mss,speed_ms,0,blend_radius_m)
      movel([0.288092, -1.467636, -2.506260, -0.738492, 1.570796, 1.858889],accel_mss,speed_ms,0,blend_radius_m)
      movel([0.287941, -1.467308, -2.506534, -0.738546, 1.570796, 1.858737],accel_mss,speed_ms,0,blend_radius_m)
      movel([0.287804, -1.466972, -2.506816, -0.738602, 1.570796, 1.858601],accel_mss,speed_ms,0,blend_radius_m)
      movel([0.287681, -1.466626, -2.507104, -0.738659, 1.570796, 1.858478],accel_mss,speed_ms,0,blend_radius_m)
      movel([0.287573, -1.466275, -2.507397, -0.738717, 1.570796, 1.858369],accel_mss,speed_ms,0,blend_radius_m)
      movel([0.287477, -1.465915, -2.507697, -0.738777, 1.570796, 1.858274],accel_mss,speed_ms,0,blend_radius_m)
      movel([0.287403, -1.465561, -2.507992, -0.738836, 1.570796, 1.858200],accel_mss,speed_ms,0,blend_radius_m)
      movel([0.287345, -1.465198, -2.508294, -0.738897, 1.570796, 1.858141],accel_mss,speed_ms,0,blend_radius_m)
      movel([0.287305, -1.464829, -2.508601, -0.738959, 1.570796, 1.858101],accel_mss,speed_ms,0,blend_radius_m)
      movel([0.287282, -1.464453, -2.508914, -0.739022, 1.570796, 1.858079],accel_mss,speed_ms,0,blend_radius_m)
      movel([0.287278, -1.464071, -2.509231, -0.739087, 1.570796, 1.858075],accel_mss,speed_ms,0,blend_radius_m)
      movel([0.287291, -1.463645, -2.509584, -0.739159, 1.570796, 1.858087],accel_mss,speed_ms,0,blend_radius_m)
      movel([0.287320, -1.463214, -2.509942, -0.739233, 1.570796, 1.858116],accel_mss,speed_ms,0,blend_radius_m)
      movel([0.287362, -1.462781, -2.510301, -0.739307, 1.570796, 1.858158],accel_mss,speed_ms,0,blend_radius_m)
      movel([0.287419, -1.462341, -2.510665, -0.739383, 1.570796, 1.858216],accel_mss,speed_ms,0,blend_radius_m)
      movel([0.287492, -1.461899, -2.511031, -0.739459, 1.570796, 1.858288],accel_mss,speed_ms,0,blend_radius_m)
      movel([0.287580, -1.461442, -2.511409, -0.739538, 1.570796, 1.858377],accel_mss,speed_ms,0,blend_radius_m)
      movel([0.287685, -1.460980, -2.511791, -0.739619, 1.570796, 1.858482],accel_mss,speed_ms,0,blend_radius_m)
      movel([0.287806, -1.460516, -2.512174, -0.739700, 1.570796, 1.858602],accel_mss,speed_ms,0,blend_radius_m)
      movel([0.287939, -1.460050, -2.512558, -0.739781, 1.570796, 1.858736],accel_mss,speed_ms,0,blend_radius_m)
      movel([0.288089, -1.459581, -2.512944, -0.739864, 1.570796, 1.858886],accel_mss,speed_ms,0,blend_radius_m)
      movel([0.288247, -1.459126, -2.513318, -0.739944, 1.570796, 1.859044],accel_mss,speed_ms,0,blend_radius_m)
      movel([0.288421, -1.458670, -2.513693, -0.740025, 1.570796, 1.859217],accel_mss,speed_ms,0,blend_radius_m)
      movel([0.288612, -1.458213, -2.514069, -0.740107, 1.570796, 1.859408],accel_mss,speed_ms,0,blend_radius_m)
      movel([0.288815, -1.457757, -2.514443, -0.740188, 1.570796, 1.859612],accel_mss,speed_ms,0,blend_radius_m)
      movel([0.289034, -1.457300, -2.514818, -0.740271, 1.570796, 1.859831],accel_mss,speed_ms,0,blend_radius_m)
      movel([0.289272, -1.456832, -2.515202, -0.740355, 1.570796, 1.860068],accel_mss,speed_ms,0,blend_radius_m)
      movel([0.289521, -1.456364, -2.515585, -0.740440, 1.570796, 1.860317],accel_mss,speed_ms,0,blend_radius_m)
      movel([0.289777, -1.455899, -2.515965, -0.740524, 1.570796, 1.860573],accel_mss,speed_ms,0,blend_radius_m)
      movel([0.290044, -1.455433, -2.516346, -0.740609, 1.570796, 1.860841],accel_mss,speed_ms,0,blend_radius_m)
      movel([0.290115, -1.455327, -2.516433, -0.740629, 1.570796, 1.860912],accel_mss,speed_ms,0,blend_radius_m)
      movel([0.290197, -1.455222, -2.516519, -0.740648, 1.570796, 1.860993],accel_mss,speed_ms,0,blend_radius_m)
      movel([0.290291, -1.455124, -2.516599, -0.740666, 1.570796, 1.861087],accel_mss,speed_ms,0,blend_radius_m)
      movel([0.290394, -1.455033, -2.516673, -0.740683, 1.570796, 1.861190],accel_mss,speed_ms,0,blend_radius_m)
      movel([0.290502, -1.454951, -2.516740, -0.740698, 1.570796, 1.861298],accel_mss,speed_ms,0,blend_radius_m)
      movel([0.290618, -1.454877, -2.516801, -0.740711, 1.570796, 1.861415],accel_mss,speed_ms,0,blend_radius_m)
      movel([0.290740, -1.454813, -2.516852, -0.740723, 1.570796, 1.861536],accel_mss,speed_ms,0,blend_radius_m)
      movel([0.290896, -1.454747, -2.516906, -0.740735, 1.570796, 1.861693],accel_mss,speed_ms,0,blend_radius_m)
      movel([0.291052, -1.454697, -2.516947, -0.740744, 1.570796, 1.861849],accel_mss,speed_ms,0,blend_radius_m)
      movel([0.291206, -1.454661, -2.516977, -0.740751, 1.570796, 1.862002],accel_mss,speed_ms,0,blend_radius_m)
      movel([0.291358, -1.454640, -2.516994, -0.740755, 1.570796, 1.862155],accel_mss,speed_ms,0,blend_radius_m)
      movel([0.291506, -1.454636, -2.516997, -0.740756, 1.570796, 1.862302],accel_mss,speed_ms,0,blend_radius_m)
      movel([0.291645, -1.454648, -2.516987, -0.740754, 1.570796, 1.862442],accel_mss,speed_ms,0,blend_radius_m)
      movel([0.292393, -1.454764, -2.516893, -0.740732, 1.570796, 1.863189],accel_mss,speed_ms,0,blend_radius_m)
      movel([0.293133, -1.454892, -2.516788, -0.740709, 1.570796, 1.863929],accel_mss,speed_ms,0,blend_radius_m)
      movel([0.293865, -1.455034, -2.516672, -0.740683, 1.570796, 1.864661],accel_mss,speed_ms,0,blend_radius_m)
      movel([0.294949, -1.455255, -2.516492, -0.740642, 1.570796, 1.865746],accel_mss,speed_ms,0,blend_radius_m)
      movel([0.295293, -1.454215, -2.517340, -0.740833, 1.570796, 1.866090],accel_mss,speed_ms,0,blend_radius_m)
      movel([0.295639, -1.453173, -2.518190, -0.741027, 1.570796, 1.866435],accel_mss,speed_ms,0,blend_radius_m)
      movel([0.271091, -1.455380, -2.516390, -0.740619, 1.570796, 1.841887],accel_mss,speed_ms,0,blend_radius_m)
      movel([0.256701, -1.456904, -2.515143, -0.740342, 1.570796, 1.827497],accel_mss,speed_ms,0,blend_radius_m)
      movel([0.253581, -1.457249, -2.514860, -0.740280, 1.570796, 1.824377],accel_mss,speed_ms,0,blend_radius_m)
      movel([0.250464, -1.457588, -2.514582, -0.740219, 1.570796, 1.821261],accel_mss,speed_ms,0,blend_radius_m)
      movel([0.248542, -1.457794, -2.514413, -0.740182, 1.570796, 1.819338],accel_mss,speed_ms,0,blend_radius_m)
      movel([0.246618, -1.457997, -2.514246, -0.740145, 1.570796, 1.817414],accel_mss,speed_ms,0,blend_radius_m)
      movel([0.246504, -1.458003, -2.514241, -0.740144, 1.570796, 1.817301],accel_mss,speed_ms,0,blend_radius_m)
      movel([0.246399, -1.457997, -2.514247, -0.740146, 1.570796, 1.817195],accel_mss,speed_ms,0,blend_radius_m)
      movel([0.246297, -1.457978, -2.514262, -0.740149, 1.570796, 1.817093],accel_mss,speed_ms,0,blend_radius_m)
      movel([0.246204, -1.457947, -2.514288, -0.740155, 1.570796, 1.817001],accel_mss,speed_ms,0,blend_radius_m)
      movel([0.246122, -1.457904, -2.514322, -0.740162, 1.570796, 1.816918],accel_mss,speed_ms,0,blend_radius_m)
      movel([0.246053, -1.457851, -2.514366, -0.740172, 1.570796, 1.816849],accel_mss,speed_ms,0,blend_radius_m)
      movel([0.246000, -1.457786, -2.514420, -0.740183, 1.570796, 1.816796],accel_mss,speed_ms,0,blend_radius_m)
      movel([0.245961, -1.457709, -2.514483, -0.740197, 1.570796, 1.816758],accel_mss,speed_ms,0,blend_radius_m)
      movel([0.245935, -1.457620, -2.514556, -0.740213, 1.570796, 1.816731],accel_mss,speed_ms,0,blend_radius_m)
      movel([0.245925, -1.457522, -2.514636, -0.740231, 1.570796, 1.816722],accel_mss,speed_ms,0,blend_radius_m)
      movel([0.245930, -1.457421, -2.514719, -0.740249, 1.570796, 1.816726],accel_mss,speed_ms,0,blend_radius_m)
      movel([0.245955, -1.457246, -2.514863, -0.740280, 1.570796, 1.816751],accel_mss,speed_ms,0,blend_radius_m)
      movel([0.245990, -1.457067, -2.515009, -0.740313, 1.570796, 1.816786],accel_mss,speed_ms,0,blend_radius_m)
      movel([0.246033, -1.456888, -2.515156, -0.740345, 1.570796, 1.816830],accel_mss,speed_ms,0,blend_radius_m)
      movel([0.246212, -1.456217, -2.515706, -0.740467, 1.570796, 1.817008],accel_mss,speed_ms,0,blend_radius_m)
      movel([0.246397, -1.455547, -2.516254, -0.740589, 1.570796, 1.817193],accel_mss,speed_ms,0,blend_radius_m)
      movel([0.247002, -1.453382, -2.518019, -0.740988, 1.570796, 1.817798],accel_mss,speed_ms,0,blend_radius_m)
      movel([0.232327, -1.455264, -2.516485, -0.740640, 1.570796, 1.803123],accel_mss,speed_ms,0,blend_radius_m)
      movel([0.217636, -1.457322, -2.514800, -0.740267, 1.570796, 1.788433],accel_mss,speed_ms,0,blend_radius_m)
      movel([0.217419, -1.458199, -2.514081, -0.740109, 1.570796, 1.788215],accel_mss,speed_ms,0,blend_radius_m)
      movel([0.217201, -1.459075, -2.513361, -0.739954, 1.570796, 1.787998],accel_mss,speed_ms,0,blend_radius_m)
      movel([0.191731, -1.463041, -2.510086, -0.739263, 1.570796, 1.762527],accel_mss,speed_ms,0,blend_radius_m)
      movel([0.166263, -1.467512, -2.506364, -0.738513, 1.570796, 1.737059],accel_mss,speed_ms,0,blend_radius_m)
      movel([0.164813, -1.468448, -2.505581, -0.738360, 1.570796, 1.735609],accel_mss,speed_ms,0,blend_radius_m)
      movel([0.164370, -1.468727, -2.505347, -0.738314, 1.570796, 1.735166],accel_mss,speed_ms,0,blend_radius_m)
      movel([0.163922, -1.468998, -2.505120, -0.738270, 1.570796, 1.734718],accel_mss,speed_ms,0,blend_radius_m)
      movel([0.163472, -1.469260, -2.504901, -0.738228, 1.570796, 1.734268],accel_mss,speed_ms,0,blend_radius_m)
      movel([0.162985, -1.469535, -2.504670, -0.738184, 1.570796, 1.733782],accel_mss,speed_ms,0,blend_radius_m)
      movel([0.162497, -1.469799, -2.504449, -0.738141, 1.570796, 1.733293],accel_mss,speed_ms,0,blend_radius_m)
      movel([0.162003, -1.470058, -2.504231, -0.738100, 1.570796, 1.732799],accel_mss,speed_ms,0,blend_radius_m)
      movel([0.161497, -1.470312, -2.504018, -0.738059, 1.570796, 1.732293],accel_mss,speed_ms,0,blend_radius_m)
      movel([0.160989, -1.470559, -2.503810, -0.738020, 1.570796, 1.731785],accel_mss,speed_ms,0,blend_radius_m)
      movel([0.160477, -1.470800, -2.503608, -0.737981, 1.570796, 1.731274],accel_mss,speed_ms,0,blend_radius_m)
      movel([0.159975, -1.471025, -2.503418, -0.737945, 1.570796, 1.730772],accel_mss,speed_ms,0,blend_radius_m)
      movel([0.159473, -1.471242, -2.503236, -0.737911, 1.570796, 1.730269],accel_mss,speed_ms,0,blend_radius_m)
      movel([0.158968, -1.471449, -2.503061, -0.737878, 1.570796, 1.729765],accel_mss,speed_ms,0,blend_radius_m)
      movel([0.158596, -1.471593, -2.502940, -0.737856, 1.570796, 1.729392],accel_mss,speed_ms,0,blend_radius_m)
      movel([0.158224, -1.471725, -2.502829, -0.737835, 1.570796, 1.729020],accel_mss,speed_ms,0,blend_radius_m)
      movel([0.157852, -1.471845, -2.502728, -0.737816, 1.570796, 1.728648],accel_mss,speed_ms,0,blend_radius_m)
      movel([0.157477, -1.471953, -2.502637, -0.737799, 1.570796, 1.728274],accel_mss,speed_ms,0,blend_radius_m)
      movel([0.156691, -1.472163, -2.502460, -0.737766, 1.570796, 1.727488],accel_mss,speed_ms,0,blend_radius_m)
      movel([0.155905, -1.472364, -2.502290, -0.737734, 1.570796, 1.726702],accel_mss,speed_ms,0,blend_radius_m)
      movel([0.155121, -1.472556, -2.502128, -0.737704, 1.570796, 1.725917],accel_mss,speed_ms,0,blend_radius_m)
      movel([0.153917, -1.472839, -2.501890, -0.737660, 1.570796, 1.724713],accel_mss,speed_ms,0,blend_radius_m)
      movel([0.152713, -1.473112, -2.501660, -0.737618, 1.570796, 1.723509],accel_mss,speed_ms,0,blend_radius_m)
      movel([0.152591, -1.473132, -2.501643, -0.737615, 1.570796, 1.723388],accel_mss,speed_ms,0,blend_radius_m)
      movel([0.152472, -1.473138, -2.501637, -0.737614, 1.570796, 1.723268],accel_mss,speed_ms,0,blend_radius_m)
      movel([0.152357, -1.473131, -2.501644, -0.737615, 1.570796, 1.723154],accel_mss,speed_ms,0,blend_radius_m)
      movel([0.152251, -1.473110, -2.501661, -0.737618, 1.570796, 1.723048],accel_mss,speed_ms,0,blend_radius_m)
      movel([0.152157, -1.473075, -2.501691, -0.737623, 1.570796, 1.722953],accel_mss,speed_ms,0,blend_radius_m)
      movel([0.152111, -1.473045, -2.501716, -0.737628, 1.570796, 1.722907],accel_mss,speed_ms,0,blend_radius_m)
      movel([0.152079, -1.473004, -2.501750, -0.737634, 1.570796, 1.722875],accel_mss,speed_ms,0,blend_radius_m)
      movel([0.152064, -1.472953, -2.501793, -0.737642, 1.570796, 1.722861],accel_mss,speed_ms,0,blend_radius_m)
      movel([0.152066, -1.472895, -2.501842, -0.737651, 1.570796, 1.722862],accel_mss,speed_ms,0,blend_radius_m)
      movel([0.152646, -1.469223, -2.504931, -0.738234, 1.570796, 1.723442],accel_mss,speed_ms,0,blend_radius_m)
      movel([0.153067, -1.466622, -2.507108, -0.738660, 1.570796, 1.723863],accel_mss,speed_ms,0,blend_radius_m)
      movel([0.153505, -1.464006, -2.509285, -0.739098, 1.570796, 1.724301],accel_mss,speed_ms,0,blend_radius_m)
      movel([0.154303, -1.459334, -2.513147, -0.739908, 1.570796, 1.725099],accel_mss,speed_ms,0,blend_radius_m)
      movel([0.155114, -1.454629, -2.517003, -0.740757, 1.570796, 1.725910],accel_mss,speed_ms,0,blend_radius_m)
      movel([0.158413, -1.435774, -2.532113, -0.744502, 1.570796, 1.729209],accel_mss,speed_ms,0,blend_radius_m)
      movel([0.159001, -1.435653, -2.532208, -0.744528, 1.570796, 1.729798],accel_mss,speed_ms,0,blend_radius_m)
      movel([0.159337, -1.435569, -2.532275, -0.744546, 1.570796, 1.730133],accel_mss,speed_ms,0,blend_radius_m)
      movel([0.159426, -1.435533, -2.532303, -0.744553, 1.570796, 1.730223],accel_mss,speed_ms,0,blend_radius_m)
      movel([0.159506, -1.435475, -2.532348, -0.744566, 1.570796, 1.730303],accel_mss,speed_ms,0,blend_radius_m)
      movel([0.159568, -1.435408, -2.532401, -0.744580, 1.570796, 1.730364],accel_mss,speed_ms,0,blend_radius_m)
      movel([0.159606, -1.435333, -2.532460, -0.744596, 1.570796, 1.730403],accel_mss,speed_ms,0,blend_radius_m)
      movel([0.159676, -1.435067, -2.532669, -0.744653, 1.570796, 1.730472],accel_mss,speed_ms,0,blend_radius_m)
      movel([0.159710, -1.434928, -2.532778, -0.744683, 1.570796, 1.730506],accel_mss,speed_ms,0,blend_radius_m)
      movel([0.159761, -1.434785, -2.532891, -0.744713, 1.570796, 1.730557],accel_mss,speed_ms,0,blend_radius_m)
      movel([0.159794, -1.434727, -2.532936, -0.744726, 1.570796, 1.730591],accel_mss,speed_ms,0,blend_radius_m)
      movel([0.159840, -1.434672, -2.532979, -0.744738, 1.570796, 1.730636],accel_mss,speed_ms,0,blend_radius_m)
      movel([0.159898, -1.434623, -2.533018, -0.744748, 1.570796, 1.730695],accel_mss,speed_ms,0,blend_radius_m)
      movel([0.159982, -1.434573, -2.533057, -0.744759, 1.570796, 1.730778],accel_mss,speed_ms,0,blend_radius_m)
      movel([0.160068, -1.434530, -2.533091, -0.744768, 1.570796, 1.730864],accel_mss,speed_ms,0,blend_radius_m)
      movel([0.160157, -1.434498, -2.533116, -0.744775, 1.570796, 1.730953],accel_mss,speed_ms,0,blend_radius_m)
      movel([0.160485, -1.434393, -2.533198, -0.744798, 1.570796, 1.731282],accel_mss,speed_ms,0,blend_radius_m)
      movel([0.160815, -1.434297, -2.533274, -0.744818, 1.570796, 1.731611],accel_mss,speed_ms,0,blend_radius_m)
      movel([0.161117, -1.434213, -2.533339, -0.744836, 1.570796, 1.731914],accel_mss,speed_ms,0,blend_radius_m)
      movel([0.161418, -1.434140, -2.533397, -0.744852, 1.570796, 1.732214],accel_mss,speed_ms,0,blend_radius_m)
      movel([0.161719, -1.434075, -2.533448, -0.744866, 1.570796, 1.732515],accel_mss,speed_ms,0,blend_radius_m)
      movel([0.162016, -1.434021, -2.533491, -0.744878, 1.570796, 1.732812],accel_mss,speed_ms,0,blend_radius_m)
      movel([0.162543, -1.433937, -2.533556, -0.744896, 1.570796, 1.733339],accel_mss,speed_ms,0,blend_radius_m)
      movel([0.163067, -1.433864, -2.533613, -0.744911, 1.570796, 1.733864],accel_mss,speed_ms,0,blend_radius_m)
      movel([0.163588, -1.433802, -2.533662, -0.744925, 1.570796, 1.734384],accel_mss,speed_ms,0,blend_radius_m)
      movel([0.164138, -1.433746, -2.533706, -0.744937, 1.570796, 1.734935],accel_mss,speed_ms,0,blend_radius_m)
      movel([0.164685, -1.433699, -2.533743, -0.744947, 1.570796, 1.735481],accel_mss,speed_ms,0,blend_radius_m)
      movel([0.165227, -1.433665, -2.533770, -0.744955, 1.570796, 1.736023],accel_mss,speed_ms,0,blend_radius_m)
      movel([0.165710, -1.433647, -2.533784, -0.744959, 1.570796, 1.736506],accel_mss,speed_ms,0,blend_radius_m)
      movel([0.166191, -1.433639, -2.533790, -0.744960, 1.570796, 1.736987],accel_mss,speed_ms,0,blend_radius_m)
      movel([0.166662, -1.433645, -2.533785, -0.744959, 1.570796, 1.737459],accel_mss,speed_ms,0,blend_radius_m)
      movel([0.167080, -1.433664, -2.533770, -0.744955, 1.570796, 1.737876],accel_mss,speed_ms,0,blend_radius_m)
      movel([0.167490, -1.433698, -2.533743, -0.744947, 1.570796, 1.738286],accel_mss,speed_ms,0,blend_radius_m)
      movel([0.167893, -1.433744, -2.533708, -0.744937, 1.570796, 1.738689],accel_mss,speed_ms,0,blend_radius_m)
      movel([0.168370, -1.433815, -2.533652, -0.744922, 1.570796, 1.739166],accel_mss,speed_ms,0,blend_radius_m)
      movel([0.168842, -1.433894, -2.533590, -0.744905, 1.570796, 1.739639],accel_mss,speed_ms,0,blend_radius_m)
      movel([0.169308, -1.433983, -2.533520, -0.744886, 1.570796, 1.740105],accel_mss,speed_ms,0,blend_radius_m)
      movel([0.169772, -1.434082, -2.533442, -0.744864, 1.570796, 1.740569],accel_mss,speed_ms,0,blend_radius_m)
      movel([0.170227, -1.434191, -2.533357, -0.744841, 1.570796, 1.741024],accel_mss,speed_ms,0,blend_radius_m)
      movel([0.170676, -1.434310, -2.533264, -0.744815, 1.570796, 1.741472],accel_mss,speed_ms,0,blend_radius_m)
      movel([0.171046, -1.434420, -2.533177, -0.744792, 1.570796, 1.741842],accel_mss,speed_ms,0,blend_radius_m)
      movel([0.171404, -1.434543, -2.533081, -0.744765, 1.570796, 1.742200],accel_mss,speed_ms,0,blend_radius_m)
      movel([0.171754, -1.434681, -2.532973, -0.744736, 1.570796, 1.742551],accel_mss,speed_ms,0,blend_radius_m)
      movel([0.172514, -1.434996, -2.532724, -0.744668, 1.570796, 1.743310],accel_mss,speed_ms,0,blend_radius_m)
      movel([0.199133, -1.430106, -2.536549, -0.745734, 1.570796, 1.769929],accel_mss,speed_ms,0,blend_radius_m)
      movel([0.225758, -1.425767, -2.539913, -0.746709, 1.570796, 1.796555],accel_mss,speed_ms,0,blend_radius_m)
      movel([0.225503, -1.426770, -2.539138, -0.746481, 1.570796, 1.796299],accel_mss,speed_ms,0,blend_radius_m)
      movel([0.225247, -1.427771, -2.538363, -0.746255, 1.570796, 1.796044],accel_mss,speed_ms,0,blend_radius_m)
      movel([0.232573, -1.426679, -2.539208, -0.746502, 1.570796, 1.803369],accel_mss,speed_ms,0,blend_radius_m)
      movel([0.237752, -1.425909, -2.539803, -0.746677, 1.570796, 1.808548],accel_mss,speed_ms,0,blend_radius_m)
      movel([0.239900, -1.425569, -2.540065, -0.746755, 1.570796, 1.810696],accel_mss,speed_ms,0,blend_radius_m)
      movel([0.239919, -1.425542, -2.540086, -0.746761, 1.570796, 1.810715],accel_mss,speed_ms,0,blend_radius_m)
      movel([0.239924, -1.425481, -2.540133, -0.746775, 1.570796, 1.810720],accel_mss,speed_ms,0,blend_radius_m)
      movel([0.239692, -1.424167, -2.541146, -0.747076, 1.570796, 1.810489],accel_mss,speed_ms,0,blend_radius_m)
      movel([0.239636, -1.423773, -2.541449, -0.747167, 1.570796, 1.810432],accel_mss,speed_ms,0,blend_radius_m)
      movel([0.239597, -1.423369, -2.541759, -0.747261, 1.570796, 1.810393],accel_mss,speed_ms,0,blend_radius_m)
      movel([0.239576, -1.422984, -2.542055, -0.747350, 1.570796, 1.810372],accel_mss,speed_ms,0,blend_radius_m)
      movel([0.239572, -1.422592, -2.542356, -0.747441, 1.570796, 1.810368],accel_mss,speed_ms,0,blend_radius_m)
      movel([0.239586, -1.422193, -2.542662, -0.747534, 1.570796, 1.810382],accel_mss,speed_ms,0,blend_radius_m)
      movel([0.239616, -1.421781, -2.542977, -0.747631, 1.570796, 1.810413],accel_mss,speed_ms,0,blend_radius_m)
      movel([0.239666, -1.421364, -2.543296, -0.747728, 1.570796, 1.810462],accel_mss,speed_ms,0,blend_radius_m)
      movel([0.239730, -1.420943, -2.543619, -0.747827, 1.570796, 1.810527],accel_mss,speed_ms,0,blend_radius_m)
      movel([0.239821, -1.420475, -2.543976, -0.747938, 1.570796, 1.810617],accel_mss,speed_ms,0,blend_radius_m)
      movel([0.239923, -1.420006, -2.544335, -0.748049, 1.570796, 1.810719],accel_mss,speed_ms,0,blend_radius_m)
      movel([0.240041, -1.419533, -2.544695, -0.748161, 1.570796, 1.810838],accel_mss,speed_ms,0,blend_radius_m)
      movel([0.240151, -1.419135, -2.544999, -0.748255, 1.570796, 1.810947],accel_mss,speed_ms,0,blend_radius_m)
      movel([0.240276, -1.418732, -2.545305, -0.748351, 1.570796, 1.811072],accel_mss,speed_ms,0,blend_radius_m)
      movel([0.240409, -1.418330, -2.545611, -0.748447, 1.570796, 1.811205],accel_mss,speed_ms,0,blend_radius_m)
      movel([0.240556, -1.417926, -2.545918, -0.748544, 1.570796, 1.811353],accel_mss,speed_ms,0,blend_radius_m)
      movel([0.240701, -1.417559, -2.546198, -0.748633, 1.570796, 1.811497],accel_mss,speed_ms,0,blend_radius_m)
      movel([0.240859, -1.417191, -2.546477, -0.748721, 1.570796, 1.811655],accel_mss,speed_ms,0,blend_radius_m)
      movel([0.241032, -1.416824, -2.546756, -0.748810, 1.570796, 1.811829],accel_mss,speed_ms,0,blend_radius_m)
      movel([0.241218, -1.416456, -2.547034, -0.748899, 1.570796, 1.812014],accel_mss,speed_ms,0,blend_radius_m)
      movel([0.241424, -1.416077, -2.547322, -0.748991, 1.570796, 1.812220],accel_mss,speed_ms,0,blend_radius_m)
      movel([0.241644, -1.415698, -2.547609, -0.749083, 1.570796, 1.812440],accel_mss,speed_ms,0,blend_radius_m)
      movel([0.241875, -1.415321, -2.547894, -0.749174, 1.570796, 1.812671],accel_mss,speed_ms,0,blend_radius_m)
      movel([0.242118, -1.414946, -2.548177, -0.749266, 1.570796, 1.812915],accel_mss,speed_ms,0,blend_radius_m)
      movel([0.242518, -1.414365, -2.548616, -0.749408, 1.570796, 1.813314],accel_mss,speed_ms,0,blend_radius_m)
      movel([0.242932, -1.413789, -2.549051, -0.749550, 1.570796, 1.813728],accel_mss,speed_ms,0,blend_radius_m)
      movel([0.243362, -1.413214, -2.549484, -0.749691, 1.570796, 1.814158],accel_mss,speed_ms,0,blend_radius_m)
      movel([0.244602, -1.411598, -2.550699, -0.750092, 1.570796, 1.815398],accel_mss,speed_ms,0,blend_radius_m)
      movel([0.242538, -1.411894, -2.550477, -0.750019, 1.570796, 1.813334],accel_mss,speed_ms,0,blend_radius_m)
      movel([0.240471, -1.412193, -2.550252, -0.749944, 1.570796, 1.811267],accel_mss,speed_ms,0,blend_radius_m)
      movel([0.240725, -1.411251, -2.550959, -0.750179, 1.570796, 1.811521],accel_mss,speed_ms,0,blend_radius_m)
      movel([0.240980, -1.410308, -2.551666, -0.750415, 1.570796, 1.811776],accel_mss,speed_ms,0,blend_radius_m)
      movel([0.234750, -1.411234, -2.550972, -0.750183, 1.570796, 1.805546],accel_mss,speed_ms,0,blend_radius_m)
      movel([0.228517, -1.412191, -2.550253, -0.749945, 1.570796, 1.799313],accel_mss,speed_ms,0,blend_radius_m)
      movel([0.228254, -1.413215, -2.549483, -0.749691, 1.570796, 1.799050],accel_mss,speed_ms,0,blend_radius_m)
      movel([0.227991, -1.414237, -2.548712, -0.749439, 1.570796, 1.798787],accel_mss,speed_ms,0,blend_radius_m)
      movel([0.200872, -1.418749, -2.545293, -0.748348, 1.570796, 1.771668],accel_mss,speed_ms,0,blend_radius_m)
      movel([0.173761, -1.423830, -2.541405, -0.747154, 1.570796, 1.744558],accel_mss,speed_ms,0,blend_radius_m)
      movel([0.171928, -1.424905, -2.540578, -0.746907, 1.570796, 1.742724],accel_mss,speed_ms,0,blend_radius_m)
      movel([0.171423, -1.425194, -2.540354, -0.746840, 1.570796, 1.742220],accel_mss,speed_ms,0,blend_radius_m)
      movel([0.170917, -1.425474, -2.540138, -0.746776, 1.570796, 1.741713],accel_mss,speed_ms,0,blend_radius_m)
      movel([0.170408, -1.425743, -2.539931, -0.746715, 1.570796, 1.741204],accel_mss,speed_ms,0,blend_radius_m)
      movel([0.169896, -1.426004, -2.539730, -0.746655, 1.570796, 1.740692],accel_mss,speed_ms,0,blend_radius_m)
      movel([0.169382, -1.426254, -2.539537, -0.746598, 1.570796, 1.740179],accel_mss,speed_ms,0,blend_radius_m)
      movel([0.168856, -1.426501, -2.539346, -0.746542, 1.570796, 1.739652],accel_mss,speed_ms,0,blend_radius_m)
      movel([0.168327, -1.426736, -2.539164, -0.746489, 1.570796, 1.739124],accel_mss,speed_ms,0,blend_radius_m)
      movel([0.167799, -1.426961, -2.538990, -0.746438, 1.570796, 1.738595],accel_mss,speed_ms,0,blend_radius_m)
      movel([0.167270, -1.427177, -2.538823, -0.746389, 1.570796, 1.738066],accel_mss,speed_ms,0,blend_radius_m)
      movel([0.166739, -1.427381, -2.538665, -0.746343, 1.570796, 1.737535],accel_mss,speed_ms,0,blend_radius_m)
      movel([0.166217, -1.427574, -2.538515, -0.746300, 1.570796, 1.737013],accel_mss,speed_ms,0,blend_radius_m)
      movel([0.165695, -1.427755, -2.538375, -0.746259, 1.570796, 1.736492],accel_mss,speed_ms,0,blend_radius_m)
      movel([0.165174, -1.427924, -2.538244, -0.746221, 1.570796, 1.735970],accel_mss,speed_ms,0,blend_radius_m)
      movel([0.164651, -1.428086, -2.538119, -0.746184, 1.570796, 1.735448],accel_mss,speed_ms,0,blend_radius_m)
      movel([0.164132, -1.428236, -2.538003, -0.746151, 1.570796, 1.734928],accel_mss,speed_ms,0,blend_radius_m)
      movel([0.163640, -1.428366, -2.537902, -0.746122, 1.570796, 1.734437],accel_mss,speed_ms,0,blend_radius_m)
      movel([0.163149, -1.428484, -2.537810, -0.746095, 1.570796, 1.733945],accel_mss,speed_ms,0,blend_radius_m)
      movel([0.162660, -1.428592, -2.537726, -0.746071, 1.570796, 1.733456],accel_mss,speed_ms,0,blend_radius_m)
      movel([0.162175, -1.428685, -2.537654, -0.746050, 1.570796, 1.732972],accel_mss,speed_ms,0,blend_radius_m)
      movel([0.161691, -1.428767, -2.537590, -0.746032, 1.570796, 1.732488],accel_mss,speed_ms,0,blend_radius_m)
      movel([0.161060, -1.428864, -2.537515, -0.746010, 1.570796, 1.731856],accel_mss,speed_ms,0,blend_radius_m)
      movel([0.160519, -1.428936, -2.537459, -0.745994, 1.570796, 1.731315],accel_mss,speed_ms,0,blend_radius_m)
      movel([0.160058, -1.428992, -2.537416, -0.745981, 1.570796, 1.730854],accel_mss,speed_ms,0,blend_radius_m)
      movel([0.160024, -1.428991, -2.537416, -0.745982, 1.570796, 1.730820],accel_mss,speed_ms,0,blend_radius_m)
      movel([0.160001, -1.428978, -2.537427, -0.745985, 1.570796, 1.730798],accel_mss,speed_ms,0,blend_radius_m)
      movel([0.159985, -1.428955, -2.537444, -0.745990, 1.570796, 1.730782],accel_mss,speed_ms,0,blend_radius_m)
      movel([0.159984, -1.428924, -2.537468, -0.745997, 1.570796, 1.730781],accel_mss,speed_ms,0,blend_radius_m)
      movel([0.160995, -1.423241, -2.541857, -0.747290, 1.570796, 1.731792],accel_mss,speed_ms,0,blend_radius_m)
      movel([0.162132, -1.416906, -2.546693, -0.748790, 1.570796, 1.732928],accel_mss,speed_ms,0,blend_radius_m)
      movel([0.163517, -1.409312, -2.552411, -0.750666, 1.570796, 1.734314],accel_mss,speed_ms,0,blend_radius_m)
      movel([0.167261, -1.389094, -2.567218, -0.756077, 1.570796, 1.738057],accel_mss,speed_ms,0,blend_radius_m)
      movel([0.167902, -1.388954, -2.567319, -0.756117, 1.570796, 1.738699],accel_mss,speed_ms,0,blend_radius_m)
      movel([0.168291, -1.388856, -2.567389, -0.756144, 1.570796, 1.739087],accel_mss,speed_ms,0,blend_radius_m)
      movel([0.168373, -1.388821, -2.567413, -0.756154, 1.570796, 1.739169],accel_mss,speed_ms,0,blend_radius_m)
      movel([0.168445, -1.388764, -2.567455, -0.756170, 1.570796, 1.739242],accel_mss,speed_ms,0,blend_radius_m)
      movel([0.168496, -1.388696, -2.567503, -0.756190, 1.570796, 1.739292],accel_mss,speed_ms,0,blend_radius_m)
      movel([0.168519, -1.388624, -2.567555, -0.756210, 1.570796, 1.739315],accel_mss,speed_ms,0,blend_radius_m)
      movel([0.168526, -1.388328, -2.567767, -0.756294, 1.570796, 1.739323],accel_mss,speed_ms,0,blend_radius_m)
      movel([0.168526, -1.388181, -2.567872, -0.756336, 1.570796, 1.739323],accel_mss,speed_ms,0,blend_radius_m)
      movel([0.168542, -1.388027, -2.567983, -0.756379, 1.570796, 1.739338],accel_mss,speed_ms,0,blend_radius_m)
      movel([0.168559, -1.387971, -2.568023, -0.756395, 1.570796, 1.739356],accel_mss,speed_ms,0,blend_radius_m)
      movel([0.168591, -1.387916, -2.568063, -0.756411, 1.570796, 1.739388],accel_mss,speed_ms,0,blend_radius_m)
      movel([0.168641, -1.387865, -2.568099, -0.756425, 1.570796, 1.739437],accel_mss,speed_ms,0,blend_radius_m)
      movel([0.168708, -1.387813, -2.568136, -0.756440, 1.570796, 1.739504],accel_mss,speed_ms,0,blend_radius_m)
      movel([0.168780, -1.387770, -2.568167, -0.756452, 1.570796, 1.739576],accel_mss,speed_ms,0,blend_radius_m)
      movel([0.168855, -1.387734, -2.568192, -0.756462, 1.570796, 1.739651],accel_mss,speed_ms,0,blend_radius_m)
      movel([0.169154, -1.387625, -2.568271, -0.756494, 1.570796, 1.739950],accel_mss,speed_ms,0,blend_radius_m)
      movel([0.169453, -1.387520, -2.568346, -0.756523, 1.570796, 1.740249],accel_mss,speed_ms,0,blend_radius_m)
      movel([0.169792, -1.387410, -2.568424, -0.756555, 1.570796, 1.740588],accel_mss,speed_ms,0,blend_radius_m)
      movel([0.170131, -1.387318, -2.568490, -0.756581, 1.570796, 1.740927],accel_mss,speed_ms,0,blend_radius_m)
      movel([0.170466, -1.387242, -2.568544, -0.756602, 1.570796, 1.741262],accel_mss,speed_ms,0,blend_radius_m)
      movel([0.170944, -1.387149, -2.568611, -0.756629, 1.570796, 1.741740],accel_mss,speed_ms,0,blend_radius_m)
      movel([0.171423, -1.387064, -2.568672, -0.756653, 1.570796, 1.742219],accel_mss,speed_ms,0,blend_radius_m)
      movel([0.171898, -1.386989, -2.568726, -0.756675, 1.570796, 1.742694],accel_mss,speed_ms,0,blend_radius_m)
      movel([0.172412, -1.386915, -2.568778, -0.756696, 1.570796, 1.743208],accel_mss,speed_ms,0,blend_radius_m)
      movel([0.172922, -1.386851, -2.568824, -0.756714, 1.570796, 1.743718],accel_mss,speed_ms,0,blend_radius_m)
      movel([0.173430, -1.386796, -2.568863, -0.756730, 1.570796, 1.744227],accel_mss,speed_ms,0,blend_radius_m)
      movel([0.173893, -1.386758, -2.568891, -0.756741, 1.570796, 1.744689],accel_mss,speed_ms,0,blend_radius_m)
      movel([0.174352, -1.386728, -2.568911, -0.756749, 1.570796, 1.745148],accel_mss,speed_ms,0,blend_radius_m)
      movel([0.174805, -1.386711, -2.568924, -0.756754, 1.570796, 1.745602],accel_mss,speed_ms,0,blend_radius_m)
      movel([0.175297, -1.386702, -2.568930, -0.756757, 1.570796, 1.746094],accel_mss,speed_ms,0,blend_radius_m)
      movel([0.175784, -1.386708, -2.568926, -0.756755, 1.570796, 1.746581],accel_mss,speed_ms,0,blend_radius_m)
      movel([0.176264, -1.386723, -2.568915, -0.756751, 1.570796, 1.747061],accel_mss,speed_ms,0,blend_radius_m)
      movel([0.176740, -1.386750, -2.568896, -0.756743, 1.570796, 1.747536],accel_mss,speed_ms,0,blend_radius_m)
      movel([0.177194, -1.386786, -2.568870, -0.756733, 1.570796, 1.747991],accel_mss,speed_ms,0,blend_radius_m)
      movel([0.177641, -1.386836, -2.568834, -0.756718, 1.570796, 1.748438],accel_mss,speed_ms,0,blend_radius_m)
      movel([0.178081, -1.386899, -2.568790, -0.756701, 1.570796, 1.748877],accel_mss,speed_ms,0,blend_radius_m)
      movel([0.178513, -1.386974, -2.568736, -0.756679, 1.570796, 1.749310],accel_mss,speed_ms,0,blend_radius_m)
      movel([0.178946, -1.387059, -2.568675, -0.756655, 1.570796, 1.749742],accel_mss,speed_ms,0,blend_radius_m)
      movel([0.179368, -1.387159, -2.568603, -0.756626, 1.570796, 1.750164],accel_mss,speed_ms,0,blend_radius_m)
      movel([0.179783, -1.387270, -2.568525, -0.756595, 1.570796, 1.750579],accel_mss,speed_ms,0,blend_radius_m)
      movel([0.180191, -1.387392, -2.568437, -0.756560, 1.570796, 1.750987],accel_mss,speed_ms,0,blend_radius_m)
      movel([0.180612, -1.387533, -2.568336, -0.756520, 1.570796, 1.751408],accel_mss,speed_ms,0,blend_radius_m)
      movel([0.181027, -1.387686, -2.568227, -0.756476, 1.570796, 1.751824],accel_mss,speed_ms,0,blend_radius_m)
      movel([0.181434, -1.387847, -2.568112, -0.756430, 1.570796, 1.752230],accel_mss,speed_ms,0,blend_radius_m)
      movel([0.181831, -1.388019, -2.567989, -0.756382, 1.570796, 1.752627],accel_mss,speed_ms,0,blend_radius_m)
      movel([0.183068, -1.388579, -2.567587, -0.756223, 1.570796, 1.753865],accel_mss,speed_ms,0,blend_radius_m)
      movel([0.210273, -1.383254, -2.571384, -0.757751, 1.570796, 1.781069],accel_mss,speed_ms,0,blend_radius_m)
      movel([0.237482, -1.378503, -2.574737, -0.759149, 1.570796, 1.808279],accel_mss,speed_ms,0,blend_radius_m)
      movel([0.237078, -1.380036, -2.573659, -0.758695, 1.570796, 1.807874],accel_mss,speed_ms,0,blend_radius_m)
      movel([0.236835, -1.381003, -2.572977, -0.758410, 1.570796, 1.807631],accel_mss,speed_ms,0,blend_radius_m)
      movel([0.236802, -1.381188, -2.572846, -0.758355, 1.570796, 1.807599],accel_mss,speed_ms,0,blend_radius_m)
      movel([0.236795, -1.381367, -2.572719, -0.758302, 1.570796, 1.807591],accel_mss,speed_ms,0,blend_radius_m)
      movel([0.236819, -1.381473, -2.572645, -0.758271, 1.570796, 1.807615],accel_mss,speed_ms,0,blend_radius_m)
      movel([0.236885, -1.381550, -2.572590, -0.758249, 1.570796, 1.807681],accel_mss,speed_ms,0,blend_radius_m)
      movel([0.236998, -1.381617, -2.572543, -0.758229, 1.570796, 1.807794],accel_mss,speed_ms,0,blend_radius_m)
      movel([0.237133, -1.381658, -2.572514, -0.758217, 1.570796, 1.807929],accel_mss,speed_ms,0,blend_radius_m)
      movel([0.237340, -1.381680, -2.572499, -0.758211, 1.570796, 1.808136],accel_mss,speed_ms,0,blend_radius_m)
      movel([0.237564, -1.381665, -2.572509, -0.758215, 1.570796, 1.808360],accel_mss,speed_ms,0,blend_radius_m)
      movel([0.246712, -1.380294, -2.573477, -0.758618, 1.570796, 1.817508],accel_mss,speed_ms,0,blend_radius_m)
      movel([0.253311, -1.379300, -2.574176, -0.758912, 1.570796, 1.824108],accel_mss,speed_ms,0,blend_radius_m)
      movel([0.269013, -1.377054, -2.575753, -0.759582, 1.570796, 1.839809],accel_mss,speed_ms,0,blend_radius_m)
      movel([0.269859, -1.374205, -2.577742, -0.760442, 1.570796, 1.840655],accel_mss,speed_ms,0,blend_radius_m)
      movel([0.270096, -1.373422, -2.578286, -0.760680, 1.570796, 1.840892],accel_mss,speed_ms,0,blend_radius_m)
      movel([0.270336, -1.372639, -2.578830, -0.760920, 1.570796, 1.841132],accel_mss,speed_ms,0,blend_radius_m)
      movel([0.270474, -1.372221, -2.579120, -0.761048, 1.570796, 1.841271],accel_mss,speed_ms,0,blend_radius_m)
      movel([0.270632, -1.371803, -2.579410, -0.761176, 1.570796, 1.841428],accel_mss,speed_ms,0,blend_radius_m)
      movel([0.270704, -1.371631, -2.579529, -0.761229, 1.570796, 1.841501],accel_mss,speed_ms,0,blend_radius_m)
      movel([0.270783, -1.371460, -2.579648, -0.761282, 1.570796, 1.841580],accel_mss,speed_ms,0,blend_radius_m)
      movel([0.270875, -1.371287, -2.579767, -0.761335, 1.570796, 1.841671],accel_mss,speed_ms,0,blend_radius_m)
      movel([0.270926, -1.371201, -2.579827, -0.761361, 1.570796, 1.841723],accel_mss,speed_ms,0,blend_radius_m)
      movel([0.270989, -1.371118, -2.579884, -0.761387, 1.570796, 1.841785],accel_mss,speed_ms,0,blend_radius_m)
      movel([0.271057, -1.371040, -2.579938, -0.761411, 1.570796, 1.841853],accel_mss,speed_ms,0,blend_radius_m)
      movel([0.271136, -1.370963, -2.579991, -0.761435, 1.570796, 1.841932],accel_mss,speed_ms,0,blend_radius_m)
      movel([0.271245, -1.370876, -2.580051, -0.761461, 1.570796, 1.842041],accel_mss,speed_ms,0,blend_radius_m)
      movel([0.271361, -1.370801, -2.580103, -0.761485, 1.570796, 1.842158],accel_mss,speed_ms,0,blend_radius_m)
      movel([0.271483, -1.370740, -2.580145, -0.761503, 1.570796, 1.842279],accel_mss,speed_ms,0,blend_radius_m)
      movel([0.271607, -1.370695, -2.580177, -0.761518, 1.570796, 1.842404],accel_mss,speed_ms,0,blend_radius_m)
      movel([0.271728, -1.370667, -2.580196, -0.761526, 1.570796, 1.842525],accel_mss,speed_ms,0,blend_radius_m)
      movel([0.273500, -1.370390, -2.580387, -0.761612, 1.570796, 1.844296],accel_mss,speed_ms,0,blend_radius_m)
      movel([0.275268, -1.370127, -2.580569, -0.761693, 1.570796, 1.846064],accel_mss,speed_ms,0,blend_radius_m)
      movel([0.278327, -1.369692, -2.580869, -0.761828, 1.570796, 1.849124],accel_mss,speed_ms,0,blend_radius_m)
      movel([0.281378, -1.369282, -2.581151, -0.761955, 1.570796, 1.852174],accel_mss,speed_ms,0,blend_radius_m)
      movel([0.298399, -1.367199, -2.582584, -0.762606, 1.570796, 1.869196],accel_mss,speed_ms,0,blend_radius_m)
      movel([0.325115, -1.364441, -2.584471, -0.763477, 1.570796, 1.895911],accel_mss,speed_ms,0,blend_radius_m)
      movel([0.326091, -1.361674, -2.586354, -0.764362, 1.570796, 1.896887],accel_mss,speed_ms,0,blend_radius_m)
      movel([0.327073, -1.358894, -2.588234, -0.765261, 1.570796, 1.897869],accel_mss,speed_ms,0,blend_radius_m)
      movel([0.310855, -1.355757, -2.590343, -0.766289, 1.570796, 1.881651],accel_mss,speed_ms,0,blend_radius_m)
      movel([0.294388, -1.352963, -2.592210, -0.767216, 1.570796, 1.865184],accel_mss,speed_ms,0,blend_radius_m)
      movel([0.294330, -1.352986, -2.592194, -0.767209, 1.570796, 1.865126],accel_mss,speed_ms,0,blend_radius_m)
      movel([0.294286, -1.353041, -2.592158, -0.767190, 1.570796, 1.865082],accel_mss,speed_ms,0,blend_radius_m)
      movel([0.292330, -1.356405, -2.589909, -0.766076, 1.570796, 1.863126],accel_mss,speed_ms,0,blend_radius_m)
      movel([0.286074, -1.358313, -2.588625, -0.765450, 1.570796, 1.856871],accel_mss,speed_ms,0,blend_radius_m)
      movel([0.283659, -1.359054, -2.588126, -0.765209, 1.570796, 1.854455],accel_mss,speed_ms,0,blend_radius_m)
      movel([0.281574, -1.359687, -2.587699, -0.765003, 1.570796, 1.852370],accel_mss,speed_ms,0,blend_radius_m)
      movel([0.279765, -1.360234, -2.587329, -0.764826, 1.570796, 1.850561],accel_mss,speed_ms,0,blend_radius_m)
      movel([0.279641, -1.360266, -2.587307, -0.764816, 1.570796, 1.850437],accel_mss,speed_ms,0,blend_radius_m)
      movel([0.279523, -1.360287, -2.587293, -0.764809, 1.570796, 1.850319],accel_mss,speed_ms,0,blend_radius_m)
      movel([0.279396, -1.360295, -2.587288, -0.764806, 1.570796, 1.850193],accel_mss,speed_ms,0,blend_radius_m)
      movel([0.279278, -1.360286, -2.587294, -0.764809, 1.570796, 1.850074],accel_mss,speed_ms,0,blend_radius_m)
      movel([0.279168, -1.360263, -2.587309, -0.764817, 1.570796, 1.849965],accel_mss,speed_ms,0,blend_radius_m)
      movel([0.270327, -1.357567, -2.589128, -0.765694, 1.570796, 1.841124],accel_mss,speed_ms,0,blend_radius_m)
      movel([0.261415, -1.354966, -2.590873, -0.766551, 1.570796, 1.832211],accel_mss,speed_ms,0,blend_radius_m)
      movel([0.261302, -1.354925, -2.590900, -0.766564, 1.570796, 1.832098],accel_mss,speed_ms,0,blend_radius_m)
      movel([0.261203, -1.354868, -2.590938, -0.766583, 1.570796, 1.831999],accel_mss,speed_ms,0,blend_radius_m)
      movel([0.261118, -1.354796, -2.590986, -0.766607, 1.570796, 1.831914],accel_mss,speed_ms,0,blend_radius_m)
      movel([0.261097, -1.354759, -2.591011, -0.766619, 1.570796, 1.831893],accel_mss,speed_ms,0,blend_radius_m)
      movel([0.261096, -1.354712, -2.591042, -0.766635, 1.570796, 1.831892],accel_mss,speed_ms,0,blend_radius_m)
      movel([0.261113, -1.354660, -2.591077, -0.766652, 1.570796, 1.831910],accel_mss,speed_ms,0,blend_radius_m)
      movel([0.263957, -1.349126, -2.594755, -0.768507, 1.570796, 1.834753],accel_mss,speed_ms,0,blend_radius_m)
      movel([0.266811, -1.343590, -2.598392, -0.770406, 1.570796, 1.837608],accel_mss,speed_ms,0,blend_radius_m)
      movel([0.266866, -1.343502, -2.598450, -0.770437, 1.570796, 1.837662],accel_mss,speed_ms,0,blend_radius_m)
      movel([0.266935, -1.343416, -2.598506, -0.770467, 1.570796, 1.837731],accel_mss,speed_ms,0,blend_radius_m)
      movel([0.267016, -1.343338, -2.598558, -0.770494, 1.570796, 1.837812],accel_mss,speed_ms,0,blend_radius_m)
      movel([0.267045, -1.343319, -2.598569, -0.770500, 1.570796, 1.837842],accel_mss,speed_ms,0,blend_radius_m)
      movel([0.267077, -1.343310, -2.598576, -0.770504, 1.570796, 1.837874],accel_mss,speed_ms,0,blend_radius_m)
      movel([0.267102, -1.343315, -2.598572, -0.770502, 1.570796, 1.837899],accel_mss,speed_ms,0,blend_radius_m)
      movel([0.268725, -1.344071, -2.598078, -0.770240, 1.570796, 1.839521],accel_mss,speed_ms,0,blend_radius_m)
      movel([0.269631, -1.344501, -2.597797, -0.770091, 1.570796, 1.840427],accel_mss,speed_ms,0,blend_radius_m)
      movel([0.270532, -1.344937, -2.597512, -0.769941, 1.570796, 1.841328],accel_mss,speed_ms,0,blend_radius_m)
      movel([0.272650, -1.345988, -2.596822, -0.769578, 1.570796, 1.843446],accel_mss,speed_ms,0,blend_radius_m)
      movel([0.278166, -1.348720, -2.595024, -0.768645, 1.570796, 1.848963],accel_mss,speed_ms,0,blend_radius_m)
      movel([0.278285, -1.348576, -2.595119, -0.768694, 1.570796, 1.849081],accel_mss,speed_ms,0,blend_radius_m)
      movel([0.278376, -1.348425, -2.595219, -0.768746, 1.570796, 1.849173],accel_mss,speed_ms,0,blend_radius_m)
      movel([0.283830, -1.337483, -2.602356, -0.772550, 1.570796, 1.854627],accel_mss,speed_ms,0,blend_radius_m)
      movel([0.283836, -1.337375, -2.602426, -0.772588, 1.570796, 1.854633],accel_mss,speed_ms,0,blend_radius_m)
      movel([0.283822, -1.337343, -2.602447, -0.772600, 1.570796, 1.854618],accel_mss,speed_ms,0,blend_radius_m)
      movel([0.283787, -1.337329, -2.602455, -0.772604, 1.570796, 1.854584],accel_mss,speed_ms,0,blend_radius_m)
      movel([0.283742, -1.337333, -2.602453, -0.772603, 1.570796, 1.854539],accel_mss,speed_ms,0,blend_radius_m)
      movel([0.278636, -1.338920, -2.601428, -0.772041, 1.570796, 1.849432],accel_mss,speed_ms,0,blend_radius_m)
      movel([0.275412, -1.339976, -2.600745, -0.771669, 1.570796, 1.846208],accel_mss,speed_ms,0,blend_radius_m)
      movel([0.272189, -1.341044, -2.600051, -0.771294, 1.570796, 1.842985],accel_mss,speed_ms,0,blend_radius_m)
      movel([0.270827, -1.341491, -2.599761, -0.771137, 1.570796, 1.841623],accel_mss,speed_ms,0,blend_radius_m)
      movel([0.269467, -1.341935, -2.599472, -0.770982, 1.570796, 1.840264],accel_mss,speed_ms,0,blend_radius_m)
      movel([0.267045, -1.342721, -2.598959, -0.770708, 1.570796, 1.837841],accel_mss,speed_ms,0,blend_radius_m)
      movel([0.267009, -1.342727, -2.598956, -0.770706, 1.570796, 1.837805],accel_mss,speed_ms,0,blend_radius_m)
      movel([0.266979, -1.342723, -2.598959, -0.770708, 1.570796, 1.837775],accel_mss,speed_ms,0,blend_radius_m)
      movel([0.266956, -1.342708, -2.598968, -0.770713, 1.570796, 1.837753],accel_mss,speed_ms,0,blend_radius_m)
      movel([0.266937, -1.342674, -2.598990, -0.770724, 1.570796, 1.837733],accel_mss,speed_ms,0,blend_radius_m)
      movel([0.266937, -1.342631, -2.599019, -0.770740, 1.570796, 1.837734],accel_mss,speed_ms,0,blend_radius_m)
      movel([0.266954, -1.342583, -2.599050, -0.770756, 1.570796, 1.837750],accel_mss,speed_ms,0,blend_radius_m)
      movel([0.269758, -1.337231, -2.602519, -0.772639, 1.570796, 1.840554],accel_mss,speed_ms,0,blend_radius_m)
      movel([0.272554, -1.331912, -2.605927, -0.774550, 1.570796, 1.843350],accel_mss,speed_ms,0,blend_radius_m)
      movel([0.272617, -1.331805, -2.605996, -0.774589, 1.570796, 1.843414],accel_mss,speed_ms,0,blend_radius_m)
      movel([0.272695, -1.331700, -2.606063, -0.774627, 1.570796, 1.843491],accel_mss,speed_ms,0,blend_radius_m)
      movel([0.272783, -1.331602, -2.606125, -0.774662, 1.570796, 1.843579],accel_mss,speed_ms,0,blend_radius_m)
      movel([0.272808, -1.331582, -2.606137, -0.774669, 1.570796, 1.843605],accel_mss,speed_ms,0,blend_radius_m)
      movel([0.272831, -1.331572, -2.606144, -0.774673, 1.570796, 1.843627],accel_mss,speed_ms,0,blend_radius_m)
      movel([0.277063, -1.330090, -2.607086, -0.775213, 1.570796, 1.847860],accel_mss,speed_ms,0,blend_radius_m)
      movel([0.281743, -1.328470, -2.608113, -0.775806, 1.570796, 1.852540],accel_mss,speed_ms,0,blend_radius_m)
      movel([0.287304, -1.326568, -2.609314, -0.776508, 1.570796, 1.858101],accel_mss,speed_ms,0,blend_radius_m)
      movel([0.301842, -1.321701, -2.612364, -0.778324, 1.570796, 1.872638],accel_mss,speed_ms,0,blend_radius_m)
      movel([0.305000, -1.325527, -2.609968, -0.776893, 1.570796, 1.875797],accel_mss,speed_ms,0,blend_radius_m)
      movel([0.308129, -1.329351, -2.607555, -0.775483, 1.570796, 1.878925],accel_mss,speed_ms,0,blend_radius_m)
      movel([0.307107, -1.331106, -2.606441, -0.774842, 1.570796, 1.877903],accel_mss,speed_ms,0,blend_radius_m)
      movel([0.306721, -1.331785, -2.606008, -0.774596, 1.570796, 1.877518],accel_mss,speed_ms,0,blend_radius_m)
      movel([0.306411, -1.332373, -2.605633, -0.774383, 1.570796, 1.877207],accel_mss,speed_ms,0,blend_radius_m)
      movel([0.306157, -1.332915, -2.605287, -0.774186, 1.570796, 1.876953],accel_mss,speed_ms,0,blend_radius_m)
      movel([0.306172, -1.332958, -2.605260, -0.774171, 1.570796, 1.876968],accel_mss,speed_ms,0,blend_radius_m)
      movel([0.306268, -1.333038, -2.605209, -0.774142, 1.570796, 1.877064],accel_mss,speed_ms,0,blend_radius_m)
      movel([0.306398, -1.333078, -2.605184, -0.774128, 1.570796, 1.877195],accel_mss,speed_ms,0,blend_radius_m)
      movel([0.311213, -1.333696, -2.604788, -0.773905, 1.570796, 1.882010],accel_mss,speed_ms,0,blend_radius_m)
      movel([0.320437, -1.334869, -2.604037, -0.773483, 1.570796, 1.891234],accel_mss,speed_ms,0,blend_radius_m)
      movel([0.323558, -1.335300, -2.603760, -0.773328, 1.570796, 1.894354],accel_mss,speed_ms,0,blend_radius_m)
      movel([0.324925, -1.335500, -2.603632, -0.773257, 1.570796, 1.895722],accel_mss,speed_ms,0,blend_radius_m)
      movel([0.326283, -1.335712, -2.603496, -0.773181, 1.570796, 1.897079],accel_mss,speed_ms,0,blend_radius_m)
      movel([0.327633, -1.335936, -2.603352, -0.773101, 1.570796, 1.898430],accel_mss,speed_ms,0,blend_radius_m)
      movel([0.328698, -1.336123, -2.603232, -0.773034, 1.570796, 1.899494],accel_mss,speed_ms,0,blend_radius_m)
      movel([0.329757, -1.336324, -2.603103, -0.772962, 1.570796, 1.900553],accel_mss,speed_ms,0,blend_radius_m)
      movel([0.330806, -1.336536, -2.602966, -0.772887, 1.570796, 1.901602],accel_mss,speed_ms,0,blend_radius_m)
      movel([0.331849, -1.336759, -2.602823, -0.772807, 1.570796, 1.902645],accel_mss,speed_ms,0,blend_radius_m)
      movel([0.332884, -1.336994, -2.602672, -0.772724, 1.570796, 1.903680],accel_mss,speed_ms,0,blend_radius_m)
      movel([0.333909, -1.337242, -2.602511, -0.772635, 1.570796, 1.904705],accel_mss,speed_ms,0,blend_radius_m)
      movel([0.334919, -1.337502, -2.602344, -0.772543, 1.570796, 1.905716],accel_mss,speed_ms,0,blend_radius_m)
      movel([0.335918, -1.337779, -2.602165, -0.772445, 1.570796, 1.906715],accel_mss,speed_ms,0,blend_radius_m)
      movel([0.336903, -1.338074, -2.601975, -0.772340, 1.570796, 1.907699],accel_mss,speed_ms,0,blend_radius_m)
      movel([0.337876, -1.338383, -2.601775, -0.772231, 1.570796, 1.908673],accel_mss,speed_ms,0,blend_radius_m)
      movel([0.338838, -1.338711, -2.601563, -0.772115, 1.570796, 1.909634],accel_mss,speed_ms,0,blend_radius_m)
      movel([0.339784, -1.339058, -2.601339, -0.771992, 1.570796, 1.910581],accel_mss,speed_ms,0,blend_radius_m)
      movel([0.340718, -1.339418, -2.601106, -0.771865, 1.570796, 1.911514],accel_mss,speed_ms,0,blend_radius_m)
      movel([0.341639, -1.339796, -2.600861, -0.771732, 1.570796, 1.912435],accel_mss,speed_ms,0,blend_radius_m)
      movel([0.342213, -1.340047, -2.600699, -0.771644, 1.570796, 1.913009],accel_mss,speed_ms,0,blend_radius_m)
      movel([0.342773, -1.340315, -2.600525, -0.771550, 1.570796, 1.913569],accel_mss,speed_ms,0,blend_radius_m)
      movel([0.343317, -1.340599, -2.600340, -0.771450, 1.570796, 1.914114],accel_mss,speed_ms,0,blend_radius_m)
      movel([0.343851, -1.340898, -2.600146, -0.771345, 1.570796, 1.914647],accel_mss,speed_ms,0,blend_radius_m)
      movel([0.344371, -1.341212, -2.599942, -0.771235, 1.570796, 1.915167],accel_mss,speed_ms,0,blend_radius_m)
      movel([0.344873, -1.341543, -2.599727, -0.771119, 1.570796, 1.915669],accel_mss,speed_ms,0,blend_radius_m)
      movel([0.345365, -1.341886, -2.599504, -0.770999, 1.570796, 1.916161],accel_mss,speed_ms,0,blend_radius_m)
      movel([0.345838, -1.342245, -2.599270, -0.770874, 1.570796, 1.916634],accel_mss,speed_ms,0,blend_radius_m)
      movel([0.346299, -1.342617, -2.599028, -0.770744, 1.570796, 1.917096],accel_mss,speed_ms,0,blend_radius_m)
      movel([0.346745, -1.343004, -2.598775, -0.770610, 1.570796, 1.917541],accel_mss,speed_ms,0,blend_radius_m)
      movel([0.347102, -1.343342, -2.598554, -0.770492, 1.570796, 1.917898],accel_mss,speed_ms,0,blend_radius_m)
      movel([0.347445, -1.343694, -2.598325, -0.770370, 1.570796, 1.918241],accel_mss,speed_ms,0,blend_radius_m)
      movel([0.347770, -1.344058, -2.598087, -0.770244, 1.570796, 1.918566],accel_mss,speed_ms,0,blend_radius_m)
      movel([0.348077, -1.344438, -2.597838, -0.770113, 1.570796, 1.918874],accel_mss,speed_ms,0,blend_radius_m)
      movel([0.348370, -1.344831, -2.597581, -0.769977, 1.570796, 1.919166],accel_mss,speed_ms,0,blend_radius_m)
      movel([0.348643, -1.345236, -2.597315, -0.769837, 1.570796, 1.919439],accel_mss,speed_ms,0,blend_radius_m)
      movel([0.348899, -1.345655, -2.597041, -0.769693, 1.570796, 1.919695],accel_mss,speed_ms,0,blend_radius_m)
      movel([0.349139, -1.346084, -2.596759, -0.769545, 1.570796, 1.919935],accel_mss,speed_ms,0,blend_radius_m)
      movel([0.349359, -1.346527, -2.596469, -0.769394, 1.570796, 1.920155],accel_mss,speed_ms,0,blend_radius_m)
      movel([0.349562, -1.346982, -2.596169, -0.769238, 1.570796, 1.920358],accel_mss,speed_ms,0,blend_radius_m)
      movel([0.349722, -1.347379, -2.595908, -0.769102, 1.570796, 1.920518],accel_mss,speed_ms,0,blend_radius_m)
      movel([0.349862, -1.347790, -2.595637, -0.768962, 1.570796, 1.920658],accel_mss,speed_ms,0,blend_radius_m)
      movel([0.349985, -1.348206, -2.595363, -0.768820, 1.570796, 1.920782],accel_mss,speed_ms,0,blend_radius_m)
      movel([0.350092, -1.348635, -2.595080, -0.768674, 1.570796, 1.920888],accel_mss,speed_ms,0,blend_radius_m)
      movel([0.350181, -1.349073, -2.594791, -0.768526, 1.570796, 1.920978],accel_mss,speed_ms,0,blend_radius_m)
      movel([0.350254, -1.349515, -2.594498, -0.768376, 1.570796, 1.921050],accel_mss,speed_ms,0,blend_radius_m)
      movel([0.350308, -1.349969, -2.594198, -0.768222, 1.570796, 1.921104],accel_mss,speed_ms,0,blend_radius_m)
      movel([0.350344, -1.350430, -2.593893, -0.768067, 1.570796, 1.921141],accel_mss,speed_ms,0,blend_radius_m)
      movel([0.350367, -1.350896, -2.593583, -0.767909, 1.570796, 1.921163],accel_mss,speed_ms,0,blend_radius_m)
      movel([0.350368, -1.351369, -2.593270, -0.767750, 1.570796, 1.921164],accel_mss,speed_ms,0,blend_radius_m)
      movel([0.350354, -1.351849, -2.592951, -0.767589, 1.570796, 1.921150],accel_mss,speed_ms,0,blend_radius_m)
      movel([0.350332, -1.352181, -2.592730, -0.767478, 1.570796, 1.921128],accel_mss,speed_ms,0,blend_radius_m)
      movel([0.350291, -1.352517, -2.592506, -0.767365, 1.570796, 1.921087],accel_mss,speed_ms,0,blend_radius_m)
      movel([0.350237, -1.352856, -2.592281, -0.767252, 1.570796, 1.921033],accel_mss,speed_ms,0,blend_radius_m)
      movel([0.350168, -1.353199, -2.592052, -0.767138, 1.570796, 1.920964],accel_mss,speed_ms,0,blend_radius_m)
      movel([0.350080, -1.353547, -2.591820, -0.767022, 1.570796, 1.920876],accel_mss,speed_ms,0,blend_radius_m)
      movel([0.349913, -1.354148, -2.591420, -0.766822, 1.570796, 1.920710],accel_mss,speed_ms,0,blend_radius_m)
      movel([0.349733, -1.354753, -2.591015, -0.766621, 1.570796, 1.920530],accel_mss,speed_ms,0,blend_radius_m)
      movel([0.349542, -1.355357, -2.590611, -0.766421, 1.570796, 1.920338],accel_mss,speed_ms,0,blend_radius_m)
      movel([0.349336, -1.355963, -2.590205, -0.766221, 1.570796, 1.920132],accel_mss,speed_ms,0,blend_radius_m)
      movel([0.349114, -1.356586, -2.589787, -0.766016, 1.570796, 1.919910],accel_mss,speed_ms,0,blend_radius_m)
      movel([0.348880, -1.357207, -2.589370, -0.765812, 1.570796, 1.919677],accel_mss,speed_ms,0,blend_radius_m)
      movel([0.348632, -1.357830, -2.588951, -0.765608, 1.570796, 1.919429],accel_mss,speed_ms,0,blend_radius_m)
      movel([0.348373, -1.358452, -2.588532, -0.765405, 1.570796, 1.919169],accel_mss,speed_ms,0,blend_radius_m)
      movel([0.348196, -1.358850, -2.588264, -0.765275, 1.570796, 1.918992],accel_mss,speed_ms,0,blend_radius_m)
      movel([0.348009, -1.359245, -2.587997, -0.765147, 1.570796, 1.918806],accel_mss,speed_ms,0,blend_radius_m)
      movel([0.347809, -1.359642, -2.587729, -0.765018, 1.570796, 1.918605],accel_mss,speed_ms,0,blend_radius_m)
      movel([0.347597, -1.360037, -2.587463, -0.764890, 1.570796, 1.918394],accel_mss,speed_ms,0,blend_radius_m)
      movel([0.347375, -1.360430, -2.587197, -0.764763, 1.570796, 1.918171],accel_mss,speed_ms,0,blend_radius_m)
      movel([0.347099, -1.360895, -2.586882, -0.764612, 1.570796, 1.917895],accel_mss,speed_ms,0,blend_radius_m)
      movel([0.346814, -1.361360, -2.586566, -0.764462, 1.570796, 1.917610],accel_mss,speed_ms,0,blend_radius_m)
      movel([0.346707, -1.361528, -2.586453, -0.764409, 1.570796, 1.917503],accel_mss,speed_ms,0,blend_radius_m)
      movel([0.346590, -1.361689, -2.586344, -0.764357, 1.570796, 1.917386],accel_mss,speed_ms,0,blend_radius_m)
      movel([0.346461, -1.361851, -2.586234, -0.764305, 1.570796, 1.917257],accel_mss,speed_ms,0,blend_radius_m)
      movel([0.346356, -1.361968, -2.586154, -0.764267, 1.570796, 1.917152],accel_mss,speed_ms,0,blend_radius_m)
      movel([0.346242, -1.362079, -2.586079, -0.764231, 1.570796, 1.917038],accel_mss,speed_ms,0,blend_radius_m)
      movel([0.346118, -1.362183, -2.586008, -0.764198, 1.570796, 1.916914],accel_mss,speed_ms,0,blend_radius_m)
      movel([0.345968, -1.362294, -2.585933, -0.764162, 1.570796, 1.916764],accel_mss,speed_ms,0,blend_radius_m)
      movel([0.345813, -1.362399, -2.585861, -0.764129, 1.570796, 1.916610],accel_mss,speed_ms,0,blend_radius_m)
      movel([0.345658, -1.362495, -2.585796, -0.764098, 1.570796, 1.916454],accel_mss,speed_ms,0,blend_radius_m)
      movel([0.345229, -1.362754, -2.585620, -0.764015, 1.570796, 1.916025],accel_mss,speed_ms,0,blend_radius_m)
      movel([0.345135, -1.362822, -2.585574, -0.763993, 1.570796, 1.915932],accel_mss,speed_ms,0,blend_radius_m)
      movel([0.345053, -1.362903, -2.585519, -0.763967, 1.570796, 1.915850],accel_mss,speed_ms,0,blend_radius_m)
      movel([0.345015, -1.362967, -2.585475, -0.763947, 1.570796, 1.915811],accel_mss,speed_ms,0,blend_radius_m)
      movel([0.345009, -1.363027, -2.585435, -0.763928, 1.570796, 1.915806],accel_mss,speed_ms,0,blend_radius_m)
      movel([0.345082, -1.363155, -2.585347, -0.763886, 1.570796, 1.915878],accel_mss,speed_ms,0,blend_radius_m)
      movel([0.345117, -1.363205, -2.585313, -0.763871, 1.570796, 1.915914],accel_mss,speed_ms,0,blend_radius_m)
      movel([0.345141, -1.363262, -2.585274, -0.763852, 1.570796, 1.915937],accel_mss,speed_ms,0,blend_radius_m)
      movel([0.345151, -1.363330, -2.585228, -0.763831, 1.570796, 1.915947],accel_mss,speed_ms,0,blend_radius_m)
      movel([0.345146, -1.363401, -2.585180, -0.763808, 1.570796, 1.915942],accel_mss,speed_ms,0,blend_radius_m)
      movel([0.345127, -1.363475, -2.585130, -0.763785, 1.570796, 1.915924],accel_mss,speed_ms,0,blend_radius_m)
      movel([0.344852, -1.364314, -2.584558, -0.763517, 1.570796, 1.915649],accel_mss,speed_ms,0,blend_radius_m)
      movel([0.344566, -1.365154, -2.583985, -0.763251, 1.570796, 1.915362],accel_mss,speed_ms,0,blend_radius_m)
      movel([0.344087, -1.366517, -2.583052, -0.762820, 1.570796, 1.914883],accel_mss,speed_ms,0,blend_radius_m)
      movel([0.343595, -1.367879, -2.582117, -0.762393, 1.570796, 1.914391],accel_mss,speed_ms,0,blend_radius_m)
      movel([0.341468, -1.373632, -2.578140, -0.760616, 1.570796, 1.912264],accel_mss,speed_ms,0,blend_radius_m)
      movel([0.337741, -1.383732, -2.571045, -0.757612, 1.570796, 1.908537],accel_mss,speed_ms,0,blend_radius_m)
      movel([0.341498, -1.383423, -2.571264, -0.757702, 1.570796, 1.912294],accel_mss,speed_ms,0,blend_radius_m)
      movel([0.345249, -1.383127, -2.571474, -0.757788, 1.570796, 1.916046],accel_mss,speed_ms,0,blend_radius_m)
      movel([0.348358, -1.376442, -2.576181, -0.759766, 1.570796, 1.919155],accel_mss,speed_ms,0,blend_radius_m)
      movel([0.349582, -1.373822, -2.578009, -0.760559, 1.570796, 1.920378],accel_mss,speed_ms,0,blend_radius_m)
      movel([0.350659, -1.371520, -2.579606, -0.761263, 1.570796, 1.921455],accel_mss,speed_ms,0,blend_radius_m)
      movel([0.351587, -1.369542, -2.580973, -0.761875, 1.570796, 1.922383],accel_mss,speed_ms,0,blend_radius_m)
      movel([0.351778, -1.369143, -2.581247, -0.761998, 1.570796, 1.922574],accel_mss,speed_ms,0,blend_radius_m)
      movel([0.351845, -1.369022, -2.581331, -0.762036, 1.570796, 1.922642],accel_mss,speed_ms,0,blend_radius_m)
      movel([0.351926, -1.368901, -2.581414, -0.762074, 1.570796, 1.922723],accel_mss,speed_ms,0,blend_radius_m)
      movel([0.352026, -1.368775, -2.581501, -0.762113, 1.570796, 1.922822],accel_mss,speed_ms,0,blend_radius_m)
      movel([0.352139, -1.368650, -2.581587, -0.762152, 1.570796, 1.922935],accel_mss,speed_ms,0,blend_radius_m)
      movel([0.352259, -1.368532, -2.581668, -0.762189, 1.570796, 1.923055],accel_mss,speed_ms,0,blend_radius_m)
      movel([0.352388, -1.368419, -2.581746, -0.762224, 1.570796, 1.923184],accel_mss,speed_ms,0,blend_radius_m)
      movel([0.352517, -1.368320, -2.581814, -0.762255, 1.570796, 1.923313],accel_mss,speed_ms,0,blend_radius_m)
      movel([0.352648, -1.368233, -2.581874, -0.762282, 1.570796, 1.923445],accel_mss,speed_ms,0,blend_radius_m)
      movel([0.352779, -1.368161, -2.581923, -0.762305, 1.570796, 1.923575],accel_mss,speed_ms,0,blend_radius_m)
      movel([0.352912, -1.368101, -2.581965, -0.762324, 1.570796, 1.923708],accel_mss,speed_ms,0,blend_radius_m)
      movel([0.353044, -1.368054, -2.581997, -0.762338, 1.570796, 1.923841],accel_mss,speed_ms,0,blend_radius_m)
      movel([0.353176, -1.368023, -2.582018, -0.762348, 1.570796, 1.923972],accel_mss,speed_ms,0,blend_radius_m)
      movel([0.353419, -1.367980, -2.582048, -0.762361, 1.570796, 1.924215],accel_mss,speed_ms,0,blend_radius_m)
      movel([0.353654, -1.367954, -2.582066, -0.762369, 1.570796, 1.924450],accel_mss,speed_ms,0,blend_radius_m)
      movel([0.353886, -1.367941, -2.582074, -0.762373, 1.570796, 1.924682],accel_mss,speed_ms,0,blend_radius_m)
      movel([0.354305, -1.367933, -2.582080, -0.762376, 1.570796, 1.925102],accel_mss,speed_ms,0,blend_radius_m)
      movel([0.354722, -1.367934, -2.582079, -0.762375, 1.570796, 1.925518],accel_mss,speed_ms,0,blend_radius_m)
      movel([0.355132, -1.367945, -2.582072, -0.762372, 1.570796, 1.925928],accel_mss,speed_ms,0,blend_radius_m)
      movel([0.358511, -1.368081, -2.581978, -0.762329, 1.570796, 1.929307],accel_mss,speed_ms,0,blend_radius_m)
      movel([0.360563, -1.368176, -2.581913, -0.762300, 1.570796, 1.931360],accel_mss,speed_ms,0,blend_radius_m)
      movel([0.362381, -1.368273, -2.581847, -0.762270, 1.570796, 1.933177],accel_mss,speed_ms,0,blend_radius_m)
      movel([0.363914, -1.368360, -2.581787, -0.762243, 1.570796, 1.934710],accel_mss,speed_ms,0,blend_radius_m)
      movel([0.364121, -1.368374, -2.581777, -0.762238, 1.570796, 1.934918],accel_mss,speed_ms,0,blend_radius_m)
      movel([0.364326, -1.368395, -2.581763, -0.762232, 1.570796, 1.935122],accel_mss,speed_ms,0,blend_radius_m)
      movel([0.364488, -1.368423, -2.581743, -0.762223, 1.570796, 1.935284],accel_mss,speed_ms,0,blend_radius_m)
      movel([0.364643, -1.368462, -2.581716, -0.762211, 1.570796, 1.935440],accel_mss,speed_ms,0,blend_radius_m)
      movel([0.364791, -1.368516, -2.581679, -0.762194, 1.570796, 1.935587],accel_mss,speed_ms,0,blend_radius_m)
      movel([0.364874, -1.368559, -2.581650, -0.762180, 1.570796, 1.935670],accel_mss,speed_ms,0,blend_radius_m)
      movel([0.364948, -1.368614, -2.581612, -0.762163, 1.570796, 1.935745],accel_mss,speed_ms,0,blend_radius_m)
      movel([0.365012, -1.368677, -2.581569, -0.762144, 1.570796, 1.935809],accel_mss,speed_ms,0,blend_radius_m)
      movel([0.365066, -1.368749, -2.581519, -0.762121, 1.570796, 1.935862],accel_mss,speed_ms,0,blend_radius_m)
      movel([0.365106, -1.368824, -2.581467, -0.762098, 1.570796, 1.935903],accel_mss,speed_ms,0,blend_radius_m)
      movel([0.365132, -1.368907, -2.581410, -0.762072, 1.570796, 1.935929],accel_mss,speed_ms,0,blend_radius_m)
      movel([0.365148, -1.368997, -2.581348, -0.762044, 1.570796, 1.935945],accel_mss,speed_ms,0,blend_radius_m)
      movel([0.365152, -1.369090, -2.581284, -0.762015, 1.570796, 1.935948],accel_mss,speed_ms,0,blend_radius_m)
      movel([0.365136, -1.369236, -2.581184, -0.761970, 1.570796, 1.935932],accel_mss,speed_ms,0,blend_radius_m)
      movel([0.365103, -1.369385, -2.581081, -0.761923, 1.570796, 1.935899],accel_mss,speed_ms,0,blend_radius_m)
      movel([0.365051, -1.369535, -2.580977, -0.761877, 1.570796, 1.935847],accel_mss,speed_ms,0,blend_radius_m)
      movel([0.364962, -1.369825, -2.580777, -0.761787, 1.570796, 1.935759],accel_mss,speed_ms,0,blend_radius_m)
      movel([0.364956, -1.369912, -2.580717, -0.761760, 1.570796, 1.935753],accel_mss,speed_ms,0,blend_radius_m)
      movel([0.364981, -1.369985, -2.580667, -0.761737, 1.570796, 1.935778],accel_mss,speed_ms,0,blend_radius_m)
      movel([0.365038, -1.370044, -2.580626, -0.761719, 1.570796, 1.935834],accel_mss,speed_ms,0,blend_radius_m)
      movel([0.365115, -1.370078, -2.580603, -0.761708, 1.570796, 1.935911],accel_mss,speed_ms,0,blend_radius_m)
      movel([0.365424, -1.370130, -2.580567, -0.761692, 1.570796, 1.936220],accel_mss,speed_ms,0,blend_radius_m)
      movel([0.365730, -1.370165, -2.580543, -0.761681, 1.570796, 1.936526],accel_mss,speed_ms,0,blend_radius_m)
      movel([0.366203, -1.370213, -2.580509, -0.761666, 1.570796, 1.937000],accel_mss,speed_ms,0,blend_radius_m)
      movel([0.366739, -1.370270, -2.580470, -0.761649, 1.570796, 1.937535],accel_mss,speed_ms,0,blend_radius_m)
      movel([0.367259, -1.370329, -2.580430, -0.761631, 1.570796, 1.938056],accel_mss,speed_ms,0,blend_radius_m)
      movel([0.367921, -1.370407, -2.580375, -0.761606, 1.570796, 1.938717],accel_mss,speed_ms,0,blend_radius_m)
      movel([0.368574, -1.370503, -2.580309, -0.761577, 1.570796, 1.939370],accel_mss,speed_ms,0,blend_radius_m)
      movel([0.369216, -1.370613, -2.580233, -0.761543, 1.570796, 1.940012],accel_mss,speed_ms,0,blend_radius_m)
      movel([0.369849, -1.370740, -2.580146, -0.761504, 1.570796, 1.940645],accel_mss,speed_ms,0,blend_radius_m)
      movel([0.370471, -1.370881, -2.580048, -0.761460, 1.570796, 1.941267],accel_mss,speed_ms,0,blend_radius_m)
      movel([0.371085, -1.371037, -2.579940, -0.761412, 1.570796, 1.941881],accel_mss,speed_ms,0,blend_radius_m)
      movel([0.371688, -1.371207, -2.579822, -0.761359, 1.570796, 1.942485],accel_mss,speed_ms,0,blend_radius_m)
      movel([0.372280, -1.371394, -2.579693, -0.761302, 1.570796, 1.943076],accel_mss,speed_ms,0,blend_radius_m)
      movel([0.372862, -1.371593, -2.579555, -0.761240, 1.570796, 1.943658],accel_mss,speed_ms,0,blend_radius_m)
      movel([0.373430, -1.371809, -2.579405, -0.761174, 1.570796, 1.944226],accel_mss,speed_ms,0,blend_radius_m)
      movel([0.374070, -1.372075, -2.579221, -0.761093, 1.570796, 1.944867],accel_mss,speed_ms,0,blend_radius_m)
      movel([0.374700, -1.372355, -2.579027, -0.761007, 1.570796, 1.945496],accel_mss,speed_ms,0,blend_radius_m)
      movel([0.375312, -1.372654, -2.578820, -0.760915, 1.570796, 1.946109],accel_mss,speed_ms,0,blend_radius_m)
      movel([0.375911, -1.372968, -2.578602, -0.760819, 1.570796, 1.946708],accel_mss,speed_ms,0,blend_radius_m)
